C05408=1029.929,82.915,-98.730,168.536,44.482,158.314
C05409=1029.936,83.164,-98.749,168.538,44.480,158.314
C05410=1029.942,83.413,-98.767,168.540,44.479,158.314
C05411=1029.948,83.662,-98.785,168.542,44.477,158.313
C05412=1029.954,83.911,-98.804,168.545,44.474,158.313
C05413=1029.960,84.161,-98.821,168.547,44.472,158.313
C05414=1029.967,84.410,-98.840,168.550,44.470,158.313
C05415=1029.972,84.659,-98.859,168.552,44.468,158.313
C05416=1029.979,84.909,-98.877,168.555,44.466,158.313
C05417=1029.984,85.157,-98.896,168.557,44.465,158.312
C05418=1029.991,85.406,-98.914,168.559,44.463,158.312
C05419=1029.997,85.656,-98.932,168.561,44.460,158.312
C05420=1030.003,85.905,-98.951,168.564,44.458,158.312
C05421=1030.010,86.154,-98.969,168.567,44.456,158.312
C05422=1030.016,86.404,-98.988,168.569,44.454,158.312
C05423=1030.022,86.654,-99.007,168.572,44.452,158.312
C05424=1030.027,86.902,-99.025,168.573,44.451,158.311
C05425=1030.034,87.151,-99.044,168.576,44.448,158.311
C05426=1030.040,87.400,-99.062,168.578,44.446,158.311
C05427=1030.046,87.650,-99.080,168.581,44.444,158.311
C05428=1030.053,87.899,-99.099,168.583,44.442,158.311
C05429=1030.059,88.148,-99.117,168.586,44.440,158.311
C05430=1030.066,88.397,-99.136,168.588,44.438,158.310
C05431=1030.071,88.647,-99.155,168.591,44.436,158.310
C05432=1030.077,88.897,-99.173,168.593,44.434,158.310
C05433=1030.084,89.146,-99.192,168.595,44.432,158.310
C05434=1030.090,89.395,-99.211,168.598,44.430,158.310
C05435=1030.096,89.643,-99.229,168.600,44.428,158.309
C05436=1030.103,89.892,-99.247,168.603,44.426,158.309
C05437=1030.108,90.142,-99.267,168.605,44.424,158.309
C05438=1030.114,90.392,-99.285,168.608,44.422,158.309
C05439=1030.120,90.641,-99.304,168.609,44.420,158.309
C05440=1030.126,90.890,-99.323,168.612,44.418,158.309
C05441=1030.132,91.140,-99.342,168.615,44.416,158.309
C05442=1030.139,91.389,-99.360,168.617,44.414,158.308
C05443=1030.145,91.638,-99.379,168.620,44.412,158.308
C05444=1030.152,91.923,-99.401,168.622,44.410,158.308
C05445=1030.158,92.208,-99.422,168.625,44.408,158.308
C05446=1030.165,92.493,-99.444,168.627,44.406,158.308
C05447=1030.173,92.778,-99.466,168.631,44.404,158.308
C05448=1030.178,93.027,-99.485,168.633,44.402,158.308
C05449=1030.185,93.277,-99.504,168.635,44.400,158.307
C05450=1030.191,93.526,-99.523,168.637,44.398,158.307
C05451=1030.197,93.775,-99.541,168.640,44.396,158.307
C05452=1030.203,94.025,-99.561,168.642,44.394,158.307
C05453=1030.209,94.274,-99.579,168.645,44.392,158.307
C05454=1030.216,94.523,-99.598,168.648,44.390,158.307
C05455=1030.221,94.772,-99.617,168.650,44.388,158.306
C05456=1030.228,95.021,-99.636,168.652,44.386,158.306
C05457=1030.233,95.271,-99.655,168.654,44.384,158.306
C05458=1030.240,95.520,-99.674,168.657,44.382,158.306
C05459=1030.245,95.769,-99.693,168.660,44.380,158.306
C05460=1030.252,96.019,-99.712,168.662,44.378,158.306
C05461=1030.258,96.268,-99.730,168.664,44.376,158.305
C05462=1030.264,96.517,-99.750,168.667,44.374,158.305
C05463=1030.271,96.766,-99.769,168.669,44.372,158.305
C05464=1030.276,97.015,-99.788,168.671,44.370,158.305
C05465=1030.283,97.264,-99.807,168.674,44.368,158.305
C05466=1030.289,97.514,-99.826,168.676,44.366,158.305
C05467=1030.295,97.763,-99.845,168.679,44.365,158.305
C05468=1030.301,98.012,-99.864,168.682,44.363,158.304
C05469=1030.307,98.261,-99.883,168.684,44.361,158.304
C05470=1030.314,98.510,-99.901,168.687,44.358,158.304
C05471=1030.319,98.759,-99.921,168.688,44.356,158.304
C05472=1030.326,99.008,-99.940,168.691,44.354,158.304
C05473=1030.332,99.258,-99.959,168.693,44.353,158.304
C05474=1030.338,99.507,-99.978,168.696,44.351,158.303
C05475=1030.344,99.756,-99.997,168.698,44.349,158.303
C05476=1030.350,100.005,-100.016,168.701,44.347,158.303
C05477=1030.356,100.254,-100.036,168.704,44.345,158.303
C05478=1030.362,100.504,-100.055,168.706,44.343,158.303
C05479=1030.368,100.754,-100.074,168.708,44.341,158.303
C05480=1030.375,101.002,-100.094,168.710,44.339,158.303
C05481=1030.381,101.252,-100.113,168.713,44.337,158.302
C05482=1030.386,101.501,-100.132,168.715,44.335,158.302
C05483=1030.393,101.750,-100.152,168.718,44.334,158.302
C05484=1030.399,101.999,-100.171,168.721,44.332,158.302
C05485=1030.404,102.249,-100.190,168.723,44.330,158.302
C05486=1030.410,102.497,-100.210,168.725,44.328,158.302
C05487=1030.417,102.746,-100.229,168.727,44.326,158.302
C05488=1030.422,102.996,-100.248,168.730,44.324,158.301
C05489=1030.428,103.245,-100.268,168.733,44.322,158.301
C05490=1030.435,103.494,-100.287,168.735,44.320,158.301
C05491=1030.441,103.743,-100.307,168.738,44.318,158.301
C05492=1030.447,103.992,-100.326,168.740,44.316,158.301
C05493=1030.453,104.242,-100.345,168.742,44.315,158.301
C05494=1030.460,104.491,-100.365,168.744,44.313,158.301
C05495=1030.465,104.740,-100.384,168.747,44.311,158.300
C05496=1030.471,104.989,-100.404,168.749,44.308,158.300
C05497=1030.477,105.238,-100.423,168.752,44.306,158.300
C05498=1030.483,105.487,-100.442,168.755,44.304,158.300
C05499=1030.489,105.736,-100.462,168.757,44.303,158.300
C05500=1030.495,105.986,-100.481,168.760,44.301,158.300
C05501=1030.502,106.235,-100.501,168.761,44.299,158.299
C05502=1030.508,106.484,-100.520,168.764,44.297,158.299
C05503=1030.514,106.733,-100.540,168.767,44.295,158.299
C05504=1030.520,106.983,-100.559,168.769,44.293,158.299
C05505=1030.526,107.231,-100.579,168.772,44.291,158.299
C05506=1030.532,107.481,-100.598,168.774,44.289,158.299
C05507=1030.538,107.729,-100.618,168.777,44.287,158.299
C05508=1030.546,108.015,-100.640,168.779,44.285,158.298
C05509=1030.552,108.300,-100.662,168.782,44.283,158.298
C05510=1030.560,108.586,-100.685,168.785,44.281,158.298
C05511=1030.566,108.871,-100.707,168.788,44.278,158.298
C05512=1030.573,109.120,-100.726,168.790,44.276,158.298
C05513=1030.579,109.368,-100.746,168.793,44.274,158.298
C05514=1030.585,109.619,-100.766,168.796,44.272,158.297
C05515=1030.591,109.867,-100.786,168.798,44.271,158.297
C05516=1030.597,110.116,-100.805,168.801,44.269,158.297
C05517=1030.603,110.365,-100.825,168.803,44.267,158.297
C05518=1030.610,110.615,-100.844,168.805,44.265,158.297
C05519=1030.616,110.864,-100.864,168.807,44.263,158.297
C05520=1030.622,111.113,-100.884,168.810,44.261,158.297
C05521=1030.627,111.362,-100.903,168.813,44.259,158.296
C05522=1030.633,111.611,-100.923,168.815,44.257,158.296
C05523=1030.640,111.861,-100.944,168.818,44.255,158.296
C05524=1030.646,112.110,-100.963,168.820,44.253,158.296
C05525=1030.652,112.359,-100.983,168.823,44.252,158.296
C05526=1030.658,112.608,-101.003,168.826,44.250,158.296
C05527=1030.663,112.857,-101.022,168.828,44.248,158.296
C05528=1030.670,113.107,-101.042,168.830,44.246,158.295
C05529=1030.676,113.356,-101.062,168.832,44.244,158.295
C05530=1030.682,113.604,-101.082,168.835,44.242,158.295
C05531=1030.688,113.854,-101.102,168.838,44.241,158.295
C05532=1030.694,114.103,-101.122,168.840,44.239,158.295
C05533=1030.699,114.352,-101.142,168.843,44.237,158.295
C05534=1030.705,114.601,-101.162,168.845,44.235,158.295
C05535=1030.711,114.850,-101.182,168.847,44.234,158.294
C05536=1030.717,115.099,-101.202,168.850,44.232,158.294
C05537=1030.724,115.349,-101.222,168.852,44.230,158.294
C05538=1030.729,115.598,-101.242,168.855,44.228,158.294
C05539=1030.735,115.847,-101.262,168.858,44.227,158.294
C05540=1030.741,116.096,-101.282,168.860,44.225,158.294
C05541=1030.748,116.345,-101.303,168.863,44.223,158.294
C05542=1030.754,116.594,-101.323,168.865,44.221,158.294
C05543=1030.759,116.843,-101.343,168.867,44.219,158.293
C05544=1030.765,117.092,-101.363,168.870,44.217,158.293
C05545=1030.771,117.342,-101.383,168.872,44.215,158.293
C05546=1030.777,117.590,-101.403,168.875,44.213,158.293
C05547=1030.783,117.840,-101.423,168.878,44.212,158.293
C05548=1030.788,118.089,-101.443,168.880,44.210,158.293
C05549=1030.795,118.338,-101.464,168.883,44.208,158.293
C05550=1030.801,118.587,-101.484,168.885,44.206,158.293
C05551=1030.807,118.836,-101.503,168.888,44.204,158.293
C05552=1030.813,119.086,-101.524,168.889,44.203,158.292
C05553=1030.819,119.335,-101.544,168.892,44.201,158.292
C05554=1030.825,119.584,-101.564,168.895,44.199,158.292
C05555=1030.831,119.833,-101.585,168.897,44.197,158.292
C05556=1030.837,120.082,-101.605,168.900,44.195,158.292
C05557=1030.843,120.331,-101.625,168.903,44.194,158.292
C05558=1030.849,120.581,-101.645,168.905,44.192,158.292
C05559=1030.855,120.829,-101.665,168.908,44.190,158.291
C05560=1030.861,121.078,-101.685,168.910,44.188,158.291
C05561=1030.867,121.328,-101.706,168.913,44.186,158.291
C05562=1030.873,121.577,-101.726,168.916,44.184,158.291
C05563=1030.879,121.826,-101.746,168.918,44.182,158.291
C05564=1030.886,122.075,-101.767,168.920,44.181,158.291
C05565=1030.892,122.324,-101.787,168.922,44.179,158.291
C05566=1030.897,122.573,-101.807,168.925,44.177,158.290
C05567=1030.904,122.822,-101.828,168.927,44.175,158.290
C05568=1030.910,123.071,-101.848,168.930,44.173,158.290
C05569=1030.916,123.320,-101.868,168.933,44.172,158.290
C05570=1030.922,123.569,-101.889,168.935,44.170,158.290
C05571=1030.928,123.818,-101.909,168.938,44.168,158.290
C05572=1030.935,124.104,-101.933,168.940,44.165,158.290
C05573=1030.942,124.388,-101.955,168.944,44.163,158.290
C05574=1030.949,124.673,-101.979,168.947,44.161,158.289
C05575=1030.956,124.959,-102.003,168.950,44.159,158.289
C05576=1030.962,125.208,-102.023,168.953,44.157,158.289
C05577=1030.968,125.457,-102.043,168.955,44.156,158.289
C05578=1030.974,125.706,-102.063,168.958,44.154,158.289
C05579=1030.980,125.955,-102.083,168.960,44.152,158.289
C05580=1030.986,126.205,-102.104,168.962,44.150,158.289
C05581=1030.993,126.453,-102.124,168.965,44.148,158.288
C05582=1030.999,126.702,-102.145,168.967,44.146,158.288
C05583=1031.004,126.951,-102.165,168.970,44.144,158.288
C05584=1031.011,127.201,-102.186,168.973,44.142,158.288
C05585=1031.017,127.450,-102.206,168.975,44.141,158.288
C05586=1031.024,127.699,-102.227,168.978,44.139,158.288
C05587=1031.029,127.948,-102.247,168.980,44.137,158.288
C05588=1031.036,128.197,-102.267,168.983,44.135,158.287
C05589=1031.042,128.446,-102.287,168.985,44.133,158.287
C05590=1031.049,128.695,-102.308,168.988,44.131,158.287
C05591=1031.054,128.944,-102.329,168.991,44.129,158.287
C05592=1031.060,129.194,-102.349,168.993,44.128,158.287
C05593=1031.066,129.442,-102.369,168.996,44.126,158.287
C05594=1031.073,129.692,-102.391,168.999,44.124,158.287
C05595=1031.079,129.940,-102.411,169.001,44.122,158.287
C05596=1031.085,130.190,-102.431,169.004,44.120,158.286
C05597=1031.092,130.438,-102.452,169.006,44.118,158.286
C05598=1031.097,130.688,-102.473,169.009,44.116,158.286
C05599=1031.103,130.937,-102.493,169.012,44.115,158.286
C05600=1031.110,131.186,-102.514,169.014,44.113,158.286
C05601=1031.115,131.435,-102.535,169.017,44.111,158.286
C05602=1031.122,131.684,-102.556,169.020,44.110,158.286
C05603=1031.127,131.933,-102.577,169.022,44.108,158.286
C05604=1031.134,132.183,-102.597,169.025,44.106,158.285
C05605=1031.139,132.431,-102.618,169.027,44.104,158.285
C05606=1031.146,132.681,-102.638,169.030,44.102,158.285
C05607=1031.151,132.929,-102.660,169.033,44.101,158.285
C05608=1031.157,133.179,-102.681,169.035,44.099,158.285
C05609=1031.163,133.427,-102.701,169.038,44.097,158.285
C05610=1031.169,133.677,-102.722,169.041,44.095,158.285
C05611=1031.176,133.925,-102.743,169.043,44.093,158.285
C05612=1031.181,134.175,-102.764,169.046,44.091,158.284
C05613=1031.187,134.423,-102.785,169.049,44.090,158.284
C05614=1031.194,134.673,-102.805,169.051,44.088,158.284
C05615=1031.199,134.922,-102.827,169.054,44.086,158.284
C05616=1031.206,135.170,-102.848,169.056,44.084,158.284
C05617=1031.211,135.420,-102.868,169.059,44.082,158.284
C05618=1031.217,135.669,-102.890,169.062,44.081,158.284
C05619=1031.224,135.918,-102.910,169.064,44.079,158.284
C05620=1031.230,136.167,-102.932,169.067,44.077,158.284
C05621=1031.236,136.416,-102.952,169.069,44.075,158.283
C05622=1031.242,136.665,-102.973,169.072,44.074,158.283
C05623=1031.248,136.914,-102.995,169.075,44.072,158.283
C05624=1031.255,137.163,-103.015,169.077,44.070,158.283
C05625=1031.260,137.412,-103.036,169.080,44.069,158.283
C05626=1031.266,137.661,-103.058,169.083,44.067,158.283
C05627=1031.272,137.910,-103.078,169.085,44.065,158.283
C05628=1031.278,138.159,-103.100,169.088,44.064,158.283
C05629=1031.284,138.408,-103.121,169.091,44.062,158.283
C05630=1031.290,138.658,-103.142,169.093,44.060,158.282
C05631=1031.297,138.906,-103.163,169.096,44.058,158.282
C05632=1031.302,139.155,-103.184,169.099,44.057,158.282
C05633=1031.308,139.405,-103.205,169.101,44.055,158.282
C05634=1031.314,139.654,-103.227,169.104,44.053,158.282
C05635=1031.320,139.902,-103.248,169.106,44.051,158.282
C05636=1031.327,140.187,-103.272,169.110,44.049,158.282
C05637=1031.334,140.473,-103.296,169.113,44.048,158.282
C05638=1031.341,140.758,-103.321,169.115,44.046,158.282
C05639=1031.347,141.042,-103.345,169.119,44.044,158.282
C05640=1031.354,141.291,-103.367,169.122,44.042,158.281
C05641=1031.360,141.541,-103.387,169.124,44.040,158.281
C05642=1031.365,141.789,-103.409,169.127,44.039,158.281
C05643=1031.371,142.039,-103.430,169.130,44.037,158.281
C05644=1031.378,142.287,-103.451,169.132,44.035,158.281
C05645=1031.384,142.536,-103.473,169.135,44.033,158.281
C05646=1031.390,142.785,-103.494,169.138,44.032,158.281
C05647=1031.396,143.034,-103.516,169.140,44.030,158.281
C05648=1031.401,143.283,-103.537,169.143,44.028,158.281
C05649=1031.407,143.533,-103.558,169.146,44.027,158.281
C05650=1031.414,143.782,-103.580,169.148,44.025,158.280
C05651=1031.420,144.030,-103.600,169.151,44.023,158.280
C05652=1031.426,144.279,-103.622,169.153,44.021,158.280
C05653=1031.432,144.528,-103.644,169.156,44.020,158.280
C05654=1031.438,144.778,-103.665,169.159,44.018,158.280
C05655=1031.444,145.026,-103.687,169.161,44.016,158.280
C05656=1031.450,145.275,-103.708,169.165,44.015,158.280
C05657=1031.456,145.525,-103.730,169.168,44.013,158.280
C05658=1031.462,145.773,-103.751,169.170,44.011,158.280
C05659=1031.469,146.022,-103.772,169.173,44.009,158.279
C05660=1031.475,146.271,-103.794,169.176,44.008,158.279
C05661=1031.481,146.520,-103.815,169.178,44.006,158.279
C05662=1031.487,146.769,-103.837,169.181,44.004,158.279
C05663=1031.493,147.018,-103.858,169.184,44.003,158.279
C05664=1031.499,147.267,-103.880,169.186,44.001,158.279
C05665=1031.505,147.517,-103.902,169.189,43.999,158.279
C05666=1031.511,147.765,-103.923,169.192,43.998,158.279
C05667=1031.517,148.014,-103.945,169.194,43.996,158.279
C05668=1031.522,148.264,-103.967,169.197,43.994,158.279
C05669=1031.528,148.513,-103.988,169.200,43.993,158.279
C05670=1031.534,148.761,-104.010,169.202,43.991,158.278
C05671=1031.540,149.011,-104.031,169.205,43.990,158.278
C05672=1031.546,149.260,-104.053,169.209,43.987,158.278
C05673=1031.553,149.508,-104.075,169.212,43.986,158.278
C05674=1031.558,149.757,-104.097,169.214,43.984,158.278
C05675=1031.565,150.006,-104.118,169.217,43.982,158.278
C05676=1031.571,150.255,-104.140,169.220,43.981,158.278
C05677=1031.576,150.505,-104.162,169.222,43.979,158.278
C05678=1031.582,150.753,-104.184,169.225,43.977,158.278
C05679=1031.588,151.002,-104.206,169.228,43.976,158.278
C05680=1031.594,151.251,-104.227,169.230,43.974,158.278
C05681=1031.600,151.500,-104.249,169.233,43.973,158.278
C05682=1031.607,151.750,-104.271,169.236,43.971,158.277
C05683=1031.613,151.998,-104.293,169.238,43.969,158.277
C05684=1031.618,152.247,-104.315,169.242,43.968,158.277
C05685=1031.624,152.496,-104.336,169.245,43.966,158.277
C05686=1031.630,152.745,-104.358,169.248,43.965,158.277
C05687=1031.637,152.994,-104.380,169.250,43.963,158.277
C05688=1031.643,153.243,-104.402,169.253,43.962,158.277
C05689=1031.649,153.492,-104.424,169.256,43.960,158.277
C05690=1031.655,153.740,-104.446,169.258,43.958,158.277
C05691=1031.660,153.990,-104.468,169.261,43.957,158.277
C05692=1031.666,154.239,-104.490,169.264,43.955,158.277
C05693=1031.673,154.488,-104.512,169.266,43.954,158.277
C05694=1031.678,154.737,-104.534,169.270,43.952,158.276
C05695=1031.685,154.986,-104.556,169.273,43.950,158.276
C05696=1031.690,155.234,-104.578,169.275,43.948,158.276
C05697=1031.697,155.483,-104.599,169.278,43.947,158.276
C05698=1031.702,155.732,-104.622,169.281,43.945,158.276
C05699=1031.708,155.982,-104.644,169.284,43.944,158.276
C05700=1031.715,156.266,-104.670,169.287,43.942,158.276
C05701=1031.722,156.551,-104.695,169.290,43.940,158.276
C05702=1031.730,156.835,-104.720,169.293,43.938,158.276
C05703=1031.736,157.120,-104.745,169.296,43.937,158.276
C05704=1031.742,157.369,-104.768,169.300,43.935,158.276
C05705=1031.748,157.618,-104.789,169.303,43.934,158.276
C05706=1031.754,157.867,-104.812,169.305,43.932,158.276
C05707=1031.761,158.116,-104.833,169.308,43.930,158.276
C05708=1031.766,158.364,-104.856,169.311,43.929,158.275
C05709=1031.772,158.614,-104.877,169.314,43.927,158.275
C05710=1031.778,158.862,-104.900,169.316,43.925,158.275
C05711=1031.784,159.112,-104.922,169.320,43.923,158.275
C05712=1031.790,159.360,-104.944,169.323,43.922,158.275
C05713=1031.796,159.609,-104.966,169.325,43.920,158.275
C05714=1031.802,159.858,-104.989,169.328,43.919,158.275
C05715=1031.808,160.107,-105.012,169.331,43.918,158.275
C05716=1031.814,160.356,-105.034,169.333,43.916,158.275
C05717=1031.820,160.605,-105.057,169.336,43.915,158.275
C05718=1031.826,160.854,-105.079,169.339,43.913,158.275
C05719=1031.831,161.104,-105.102,169.342,43.912,158.275
C05720=1031.837,161.352,-105.124,169.345,43.910,158.275
C05721=1031.843,161.601,-105.147,169.348,43.909,158.275
C05722=1031.848,161.849,-105.170,169.351,43.908,158.275
C05723=1031.854,162.099,-105.192,169.354,43.906,158.275
C05724=1031.860,162.348,-105.214,169.357,43.905,158.275
C05725=1031.866,162.596,-105.237,169.359,43.903,158.275
C05726=1031.872,162.845,-105.260,169.362,43.902,158.275
C05727=1031.877,163.094,-105.283,169.365,43.900,158.274
C05728=1031.884,163.343,-105.305,169.368,43.899,158.274
C05729=1031.889,163.592,-105.328,169.371,43.898,158.275
C05730=1031.895,163.841,-105.351,169.374,43.896,158.274
C05731=1031.901,164.090,-105.373,169.377,43.895,158.274
C05732=1031.907,164.339,-105.396,169.380,43.893,158.274
C05733=1031.913,164.588,-105.419,169.382,43.892,158.274
C05734=1031.918,164.837,-105.441,169.385,43.890,158.274
C05735=1031.924,165.086,-105.464,169.388,43.889,158.274
C05736=1031.931,165.335,-105.486,169.392,43.888,158.274
C05737=1031.936,165.583,-105.509,169.395,43.886,158.274
C05738=1031.942,165.832,-105.532,169.397,43.884,158.274
C05739=1031.948,166.081,-105.555,169.400,43.883,158.274
C05740=1031.954,166.330,-105.577,169.403,43.882,158.274
C05741=1031.960,166.579,-105.600,169.405,43.880,158.274
C05742=1031.966,166.828,-105.623,169.409,43.879,158.274
C05743=1031.971,167.077,-105.646,169.412,43.878,158.274
C05744=1031.978,167.325,-105.669,169.415,43.876,158.274
C05745=1031.983,167.575,-105.691,169.417,43.874,158.274
C05746=1031.989,167.824,-105.714,169.420,43.873,158.274
C05747=1031.995,168.072,-105.737,169.424,43.872,158.274
C05748=1032.001,168.321,-105.759,169.427,43.870,158.274
C05749=1032.007,168.570,-105.782,169.429,43.869,158.274
C05750=1032.013,168.819,-105.805,169.432,43.867,158.274
C05751=1032.018,169.068,-105.828,169.435,43.866,158.274
C05752=1032.025,169.317,-105.851,169.439,43.864,158.274
C05753=1032.031,169.566,-105.874,169.442,43.863,158.274
C05754=1032.037,169.814,-105.897,169.444,43.862,158.274
C05755=1032.043,170.063,-105.920,169.447,43.861,158.274
C05756=1032.049,170.312,-105.943,169.450,43.859,158.273
C05757=1032.055,170.561,-105.966,169.454,43.857,158.273
C05758=1032.061,170.809,-105.988,169.456,43.856,158.273
C05759=1032.067,171.058,-106.011,169.459,43.855,158.273
C05760=1032.073,171.308,-106.035,169.462,43.853,158.273
C05761=1032.079,171.557,-106.058,169.466,43.852,158.273
C05762=1032.085,171.805,-106.080,169.468,43.850,158.273
C05763=1032.091,172.054,-106.103,169.471,43.849,158.273
C05764=1032.098,172.338,-106.129,169.475,43.847,158.273
C05765=1032.104,172.623,-106.156,169.479,43.846,158.273
C05766=1032.111,172.907,-106.182,169.481,43.844,158.273
C05767=1032.119,173.191,-106.208,169.485,43.842,158.273
C05768=1032.124,173.439,-106.231,169.488,43.841,158.273
C05769=1032.130,173.688,-106.254,169.492,43.839,158.273
C05770=1032.136,173.938,-106.278,169.494,43.838,158.273
C05771=1032.143,174.187,-106.300,169.497,43.837,158.273
C05772=1032.149,174.435,-106.324,169.500,43.835,158.273
C05773=1032.155,174.684,-106.347,169.504,43.833,158.273
C05774=1032.160,174.933,-106.370,169.506,43.832,158.273
C05775=1032.167,175.182,-106.393,169.509,43.831,158.273
C05776=1032.173,175.431,-106.415,169.513,43.830,158.273
C05777=1032.179,175.679,-106.439,169.516,43.828,158.273
C05778=1032.185,175.928,-106.462,169.519,43.826,158.273
C05779=1032.191,176.178,-106.485,169.522,43.825,158.273
C05780=1032.197,176.426,-106.509,169.525,43.824,158.273
C05781=1032.203,176.675,-106.532,169.528,43.822,158.273
C05782=1032.210,176.924,-106.554,169.531,43.821,158.273
C05783=1032.216,177.173,-106.577,169.534,43.819,158.273
C05784=1032.222,177.421,-106.601,169.537,43.818,158.273
C05785=1032.228,177.670,-106.624,169.540,43.817,158.273
C05786=1032.234,177.920,-106.647,169.544,43.815,158.273
C05787=1032.241,178.168,-106.670,169.547,43.814,158.273
C05788=1032.247,178.417,-106.693,169.549,43.812,158.273
C05789=1032.253,178.666,-106.717,169.553,43.811,158.273
C05790=1032.259,178.914,-106.740,169.556,43.810,158.273
C05791=1032.265,179.163,-106.763,169.559,43.808,158.272
C05792=1032.271,179.412,-106.787,169.562,43.806,158.273
C05793=1032.278,179.661,-106.810,169.565,43.805,158.273
C05794=1032.284,179.909,-106.833,169.569,43.804,158.273
C05795=1032.290,180.159,-106.857,169.572,43.803,158.273
C05796=1032.296,180.408,-106.880,169.574,43.801,158.272
C05797=1032.302,180.656,-106.903,169.578,43.799,158.272
C05798=1032.308,180.906,-106.927,169.581,43.798,158.272
C05799=1032.315,181.154,-106.950,169.584,43.797,158.272
C05800=1032.321,181.403,-106.973,169.588,43.796,158.272
C05801=1032.327,181.651,-106.997,169.590,43.794,158.272
C05802=1032.333,181.900,-107.020,169.594,43.792,158.272
C05803=1032.340,182.149,-107.044,169.597,43.791,158.272
C05804=1032.345,182.398,-107.066,169.600,43.790,158.272
C05805=1032.352,182.647,-107.091,169.604,43.788,158.272
C05806=1032.359,182.896,-107.113,169.606,43.787,158.272
C05807=1032.364,183.145,-107.137,169.610,43.785,158.272
C05808=1032.370,183.393,-107.161,169.613,43.784,158.272
C05809=1032.376,183.642,-107.184,169.616,43.783,158.272
C05810=1032.381,183.891,-107.208,169.620,43.782,158.272
C05811=1032.388,184.140,-107.232,169.623,43.781,158.272
C05812=1032.393,184.388,-107.257,169.625,43.780,158.272
C05813=1032.400,184.638,-107.280,169.628,43.778,158.272
C05814=1032.406,184.886,-107.304,169.632,43.777,158.272
C05815=1032.411,185.135,-107.328,169.635,43.776,158.272
C05816=1032.418,185.384,-107.352,169.638,43.775,158.273
C05817=1032.423,185.632,-107.376,169.642,43.774,158.273
C05818=1032.429,185.881,-107.400,169.645,43.773,158.273
C05819=1032.435,186.131,-107.424,169.647,43.771,158.273
C05820=1032.441,186.379,-107.447,169.651,43.770,158.273
C05821=1032.447,186.628,-107.472,169.654,43.769,158.273
C05822=1032.453,186.876,-107.496,169.658,43.768,158.273
C05823=1032.459,187.125,-107.519,169.661,43.767,158.273
C05824=1032.465,187.374,-107.544,169.664,43.766,158.273
C05825=1032.471,187.622,-107.568,169.668,43.764,158.273
C05826=1032.477,187.872,-107.592,169.670,43.763,158.273
C05827=1032.482,188.120,-107.615,169.673,43.762,158.273
C05828=1032.489,188.404,-107.643,169.677,43.760,158.273
C05829=1032.496,188.687,-107.671,169.681,43.759,158.273
C05830=1032.502,188.972,-107.698,169.685,43.758,158.273
C05831=1032.510,189.256,-107.726,169.689,43.757,158.273
C05832=1032.516,189.504,-107.749,169.692,43.756,158.273
C05833=1032.521,189.753,-107.774,169.695,43.754,158.273
C05834=1032.528,190.002,-107.798,169.698,43.753,158.273
C05835=1032.533,190.250,-107.822,169.701,43.752,158.273
C05836=1032.539,190.499,-107.846,169.705,43.751,158.273
C05837=1032.545,190.748,-107.870,169.708,43.750,158.273
C05838=1032.551,190.997,-107.894,169.712,43.748,158.273
C05839=1032.557,191.246,-107.919,169.715,43.747,158.273
C05840=1032.563,191.494,-107.942,169.718,43.746,158.273
C05841=1032.570,191.743,-107.966,169.721,43.745,158.274
C05842=1032.576,191.991,-107.991,169.724,43.744,158.274
C05843=1032.582,192.240,-108.015,169.728,43.743,158.274
C05844=1032.588,192.489,-108.040,169.731,43.741,158.274
C05845=1032.594,192.738,-108.064,169.735,43.740,158.274
C05846=1032.599,192.986,-108.088,169.738,43.739,158.274
C05847=1032.606,193.235,-108.112,169.742,43.738,158.274
C05848=1032.612,193.485,-108.137,169.744,43.737,158.274
C05849=1032.618,193.733,-108.160,169.748,43.735,158.274
C05850=1032.624,193.982,-108.186,169.751,43.735,158.274
C05851=1032.630,194.230,-108.209,169.755,43.733,158.274
C05852=1032.636,194.479,-108.234,169.758,43.732,158.274
C05853=1032.643,194.728,-108.258,169.761,43.731,158.274
C05854=1032.648,194.977,-108.282,169.765,43.730,158.274
C05855=1032.655,195.225,-108.307,169.768,43.729,158.274
C05856=1032.660,195.474,-108.331,169.772,43.728,158.274
C05857=1032.667,195.723,-108.355,169.774,43.726,158.274
C05858=1032.673,195.972,-108.380,169.778,43.726,158.274
C05859=1032.679,196.220,-108.404,169.781,43.724,158.274
C05860=1032.685,196.469,-108.429,169.785,43.723,158.274
C05861=1032.692,196.718,-108.453,169.788,43.722,158.274
C05862=1032.697,196.967,-108.477,169.792,43.721,158.275
C05863=1032.704,197.215,-108.502,169.795,43.720,158.275
C05864=1032.710,197.464,-108.527,169.799,43.718,158.275
C05865=1032.716,197.712,-108.550,169.803,43.718,158.275
C05866=1032.722,197.961,-108.576,169.805,43.716,158.275
C05867=1032.729,198.210,-108.600,169.809,43.715,158.275
C05868=1032.735,198.459,-108.624,169.812,43.715,158.275
C05869=1032.741,198.707,-108.649,169.816,43.713,158.275
C05870=1032.747,198.956,-108.673,169.819,43.712,158.275
C05871=1032.754,199.205,-108.698,169.823,43.711,158.275
C05872=1032.760,199.454,-108.723,169.826,43.710,158.275
C05873=1032.766,199.702,-108.746,169.830,43.709,158.275
C05874=1032.772,199.951,-108.772,169.832,43.707,158.275
C05875=1032.779,200.200,-108.796,169.837,43.707,158.275
C05876=1032.785,200.449,-108.821,169.840,43.705,158.275
C05877=1032.790,200.697,-108.845,169.843,43.705,158.276
C05878=1032.796,200.946,-108.870,169.847,43.703,158.276
C05879=1032.803,201.195,-108.895,169.850,43.703,158.276
C05880=1032.809,201.443,-108.920,169.854,43.701,158.276
C05881=1032.815,201.691,-108.945,169.857,43.701,158.276
C05882=1032.821,201.941,-108.969,169.861,43.699,158.276
C05883=1032.827,202.189,-108.995,169.864,43.699,158.276
C05884=1032.833,202.439,-109.019,169.868,43.697,158.276
C05885=1032.838,202.687,-109.044,169.871,43.697,158.276
C05886=1032.845,202.935,-109.070,169.875,43.695,158.276
C05887=1032.851,203.184,-109.094,169.879,43.695,158.276
C05888=1032.858,203.433,-109.119,169.882,43.693,158.276
C05889=1032.864,203.682,-109.144,169.886,43.693,158.277
C05890=1032.869,203.930,-109.169,169.888,43.692,158.277
C05891=1032.875,204.179,-109.194,169.893,43.691,158.277
C05892=1032.901,205.228,-109.300,170.230,43.795,158.327
C05893=1032.911,205.577,-109.337,170.234,43.794,158.327
C05894=1032.921,205.926,-109.374,170.237,43.795,158.327
C05895=1032.930,206.275,-109.410,170.241,43.794,158.328
C05896=1032.940,206.624,-109.448,170.244,43.794,158.328
C05897=1032.946,206.873,-109.475,170.246,43.794,158.328
C05898=1032.953,207.121,-109.501,170.249,43.793,158.328
C05899=1032.960,207.370,-109.527,170.251,43.793,158.328
C05900=1032.966,207.618,-109.553,170.255,43.793,158.329
C05901=1032.973,207.867,-109.580,170.257,43.793,158.329
C05902=1032.980,208.116,-109.606,170.260,43.793,158.329
C05903=1032.986,208.364,-109.633,170.262,43.792,158.329
C05904=1032.994,208.612,-109.659,170.264,43.793,158.329
C05905=1032.999,208.861,-109.686,170.267,43.792,158.330
C05906=1033.006,209.110,-109.712,170.270,43.792,158.330
C05907=1033.014,209.358,-109.738,170.273,43.792,158.330
C05908=1033.020,209.606,-109.765,170.275,43.792,158.330
C05909=1033.027,209.855,-109.792,170.278,43.791,158.330
C05910=1033.034,210.104,-109.819,170.280,43.792,158.331
C05911=1033.040,210.352,-109.845,170.282,43.791,158.331
C05912=1033.047,210.601,-109.872,170.285,43.791,158.331
C05913=1033.054,210.849,-109.898,170.287,43.791,158.331
C05914=1033.061,211.097,-109.925,170.291,43.790,158.331
C05915=1033.067,211.346,-109.952,170.293,43.791,158.331
C05916=1033.074,211.595,-109.978,170.296,43.791,158.332
C05917=1033.080,211.843,-110.005,170.298,43.790,158.332
C05918=1033.087,212.091,-110.032,170.301,43.790,158.332
C05919=1033.093,212.340,-110.059,170.303,43.790,158.332
C05920=1033.100,212.588,-110.085,170.307,43.790,158.332
C05921=1033.107,212.837,-110.113,170.309,43.790,158.333
C05922=1033.113,213.085,-110.139,170.311,43.790,158.333
C05923=1033.120,213.334,-110.166,170.314,43.789,158.333
C05924=1033.127,213.582,-110.193,170.316,43.790,158.333
C05925=1033.134,213.831,-110.220,170.319,43.790,158.333
C05926=1033.140,214.079,-110.246,170.321,43.789,158.334
C05927=1033.147,214.328,-110.274,170.325,43.789,158.334
C05928=1033.154,214.576,-110.300,170.327,43.789,158.334
C05929=1033.160,214.825,-110.327,170.330,43.789,158.334
C05930=1033.167,215.073,-110.354,170.332,43.789,158.334
C05931=1033.173,215.322,-110.381,170.335,43.789,158.335
C05932=1033.181,215.570,-110.408,170.338,43.789,158.335
C05933=1033.187,215.818,-110.435,170.341,43.788,158.335
C05934=1033.194,216.067,-110.461,170.343,43.789,158.335
C05935=1033.200,216.316,-110.489,170.346,43.788,158.335
C05936=1033.208,216.564,-110.516,170.348,43.788,158.336
C05937=1033.214,216.812,-110.543,170.351,43.788,158.336
C05938=1033.221,217.061,-110.569,170.353,43.788,158.336
C05939=1033.227,217.309,-110.597,170.357,43.788,158.336
C05940=1033.235,217.558,-110.623,170.359,43.788,158.336
C05941=1033.241,217.806,-110.651,170.362,43.788,158.337
C05942=1033.248,218.054,-110.677,170.364,43.787,158.337
C05943=1033.254,218.303,-110.705,170.367,43.787,158.337
C05944=1033.262,218.552,-110.731,170.369,43.787,158.337
C05945=1033.268,218.800,-110.759,170.373,43.787,158.337
C05946=1033.275,219.048,-110.785,170.375,43.787,158.338
C05947=1033.281,219.297,-110.813,170.378,43.787,158.338
C05948=1033.289,219.545,-110.839,170.380,43.787,158.338
C05949=1033.297,219.900,-110.878,170.384,43.787,158.338
C05950=1033.307,220.255,-110.917,170.389,43.787,158.339
C05951=1033.317,220.609,-110.957,170.392,43.787,158.339
C05952=1033.326,220.964,-110.996,170.396,43.787,158.339
C05953=1033.333,221.213,-111.023,170.398,43.786,158.339
C05954=1033.339,221.461,-111.050,170.401,43.786,158.340
C05955=1033.346,221.710,-111.078,170.404,43.787,158.340
C05956=1033.353,221.958,-111.105,170.407,43.786,158.340
C05957=1033.359,222.207,-111.132,170.410,43.786,158.340
C05958=1033.366,222.455,-111.160,170.412,43.786,158.341
C05959=1033.372,222.703,-111.187,170.416,43.786,158.341
C05960=1033.379,222.951,-111.215,170.418,43.786,158.341
C05961=1033.386,223.200,-111.241,170.421,43.786,158.341
C05962=1033.393,223.449,-111.269,170.423,43.786,158.342
C05963=1033.399,223.697,-111.297,170.426,43.786,158.342
C05964=1033.406,223.945,-111.324,170.428,43.786,158.342
C05965=1033.413,224.194,-111.352,170.432,43.786,158.342
C05966=1033.420,224.443,-111.378,170.435,43.786,158.343
C05967=1033.426,224.690,-111.406,170.437,43.786,158.343
C05968=1033.432,224.939,-111.433,170.440,43.786,158.343
C05969=1033.439,225.187,-111.461,170.442,43.786,158.343
C05970=1033.446,225.436,-111.489,170.445,43.785,158.343
C05971=1033.453,225.684,-111.515,170.448,43.786,158.344
C05972=1033.460,225.933,-111.543,170.451,43.786,158.344
C05973=1033.466,226.181,-111.571,170.454,43.786,158.344
C05974=1033.473,226.430,-111.599,170.456,43.785,158.344
C05975=1033.480,226.678,-111.626,170.460,43.786,158.344
C05976=1033.486,226.927,-111.654,170.462,43.786,158.345
C05977=1033.494,227.175,-111.681,170.465,43.785,158.345
C05978=1033.500,227.423,-111.709,170.468,43.785,158.345
C05979=1033.507,227.672,-111.737,170.470,43.785,158.345
C05980=1033.514,227.920,-111.764,170.474,43.786,158.346
C05981=1033.520,228.168,-111.792,170.476,43.785,158.346
C05982=1033.527,228.416,-111.819,170.479,43.785,158.346
C05983=1033.533,228.665,-111.847,170.482,43.785,158.346
C05984=1033.540,228.913,-111.875,170.484,43.786,158.347
C05985=1033.547,229.162,-111.903,170.488,43.786,158.347
C05986=1033.553,229.410,-111.930,170.490,43.786,158.347
C05987=1033.560,229.659,-111.958,170.493,43.785,158.347
C05988=1033.567,229.907,-111.986,170.496,43.785,158.348
C05989=1033.573,230.155,-112.014,170.498,43.786,158.348
C05990=1033.580,230.404,-112.041,170.502,43.786,158.348
C05991=1033.587,230.652,-112.069,170.504,43.786,158.348
C05992=1033.593,230.901,-112.097,170.507,43.786,158.349
C05993=1033.600,231.149,-112.125,170.510,43.785,158.349
C05994=1033.607,231.397,-112.153,170.513,43.786,158.349
C05995=1033.613,231.646,-112.181,170.516,43.786,158.349
C05996=1033.620,231.894,-112.209,170.519,43.786,158.350
C05997=1033.626,232.143,-112.237,170.521,43.786,158.350
C05998=1033.633,232.390,-112.265,170.525,43.786,158.350
C05999=1033.640,232.639,-112.293,170.527,43.786,158.350
C06000=1033.646,232.888,-112.321,170.530,43.786,158.351
C06001=1033.653,233.136,-112.349,170.533,43.786,158.351
C06002=1033.659,233.385,-112.377,170.536,43.787,158.351
C06003=1033.666,233.632,-112.405,170.539,43.787,158.351
C06004=1033.673,233.881,-112.433,170.542,43.786,158.352
C06005=1033.682,234.228,-112.473,170.545,43.787,158.352
C06006=1033.691,234.575,-112.512,170.550,43.787,158.352
C06007=1033.700,234.923,-112.551,170.554,43.786,158.353
C06008=1033.709,235.270,-112.590,170.557,43.787,158.353
C06009=1033.716,235.518,-112.618,170.561,43.787,158.353
C06010=1033.724,235.767,-112.646,170.564,43.787,158.354
C06011=1033.730,236.015,-112.674,170.566,43.787,158.354
C06012=1033.737,236.263,-112.703,170.569,43.787,158.354
C06013=1033.743,236.512,-112.731,170.573,43.787,158.354
C06014=1033.750,236.760,-112.759,170.576,43.787,158.355
C06015=1033.757,237.008,-112.787,170.578,43.787,158.355
C06016=1033.763,237.257,-112.815,170.581,43.787,158.355
C06017=1033.770,237.505,-112.844,170.585,43.787,158.356
C06018=1033.777,237.753,-112.872,170.587,43.788,158.356
C06019=1033.784,238.002,-112.900,170.590,43.788,158.356
C06020=1033.790,238.250,-112.929,170.593,43.788,158.356
C06021=1033.797,238.498,-112.957,170.596,43.788,158.357
C06022=1033.804,238.747,-112.985,170.599,43.788,158.357
C06023=1033.810,238.995,-113.014,170.602,43.788,158.357
C06024=1033.817,239.243,-113.042,170.605,43.788,158.357
C06025=1033.824,239.491,-113.070,170.608,43.788,158.358
C06026=1033.831,239.740,-113.098,170.611,43.788,158.358
C06027=1033.837,239.988,-113.127,170.614,43.788,158.358
C06028=1033.844,240.237,-113.155,170.616,43.789,158.359
C06029=1033.851,240.484,-113.183,170.620,43.789,158.359
C06030=1033.857,240.733,-113.212,170.623,43.789,158.359
C06031=1033.864,240.981,-113.240,170.626,43.789,158.359
C06032=1033.870,241.229,-113.269,170.628,43.789,158.360
C06033=1033.878,241.478,-113.298,170.632,43.789,158.360
C06034=1033.884,241.726,-113.326,170.635,43.789,158.360
C06035=1033.891,241.974,-113.355,170.637,43.789,158.360
C06036=1033.897,242.222,-113.384,170.641,43.790,158.361
C06037=1033.904,242.470,-113.412,170.644,43.790,158.361
C06038=1033.910,242.720,-113.441,170.647,43.790,158.361
C06039=1033.917,242.968,-113.470,170.649,43.790,158.362
C06040=1033.924,243.216,-113.498,170.653,43.791,158.362
C06041=1033.930,243.464,-113.528,170.656,43.791,158.362
C06042=1033.937,243.712,-113.555,170.658,43.791,158.363
C06043=1033.943,243.961,-113.585,170.662,43.791,158.363
C06044=1033.950,244.209,-113.613,170.665,43.792,158.363
C06045=1033.957,244.457,-113.642,170.668,43.792,158.364
C06046=1033.964,244.705,-113.671,170.671,43.792,158.364
C06047=1033.970,244.954,-113.699,170.674,43.792,158.364
C06048=1033.976,245.202,-113.728,170.677,43.792,158.364
C06049=1033.983,245.451,-113.757,170.681,43.793,158.365
C06050=1033.989,245.699,-113.786,170.683,43.793,158.365
C06051=1033.996,245.946,-113.815,170.686,43.793,158.365
C06052=1034.002,246.195,-113.844,170.689,43.793,158.366
C06053=1034.009,246.443,-113.873,170.692,43.794,158.366
C06054=1034.015,246.692,-113.902,170.695,43.794,158.366
C06055=1034.022,246.940,-113.931,170.698,43.794,158.367
C06056=1034.029,247.188,-113.960,170.702,43.794,158.367
C06057=1034.035,247.436,-113.989,170.704,43.795,158.367
C06058=1034.042,247.684,-114.018,170.707,43.795,158.368
C06059=1034.048,247.933,-114.047,170.711,43.795,158.368
C06060=1034.054,248.181,-114.076,170.714,43.795,158.368
C06061=1034.063,248.522,-114.116,170.718,43.795,158.369
C06062=1034.073,248.863,-114.156,170.722,43.796,158.369
C06063=1034.082,249.204,-114.196,170.726,43.797,158.370
C06064=1034.091,249.546,-114.236,170.731,43.797,158.370
C06065=1034.098,249.795,-114.265,170.734,43.797,158.370
C06066=1034.104,250.043,-114.295,170.737,43.797,158.371
C06067=1034.110,250.290,-114.324,170.740,43.797,158.371
C06068=1034.117,250.539,-114.354,170.743,43.798,158.371
C06069=1034.124,250.787,-114.382,170.746,43.798,158.372
C06070=1034.130,251.035,-114.411,170.750,43.798,158.372
C06071=1034.137,251.284,-114.441,170.753,43.799,158.372
C06072=1034.144,251.532,-114.470,170.755,43.799,158.373
C06073=1034.150,251.779,-114.499,170.759,43.799,158.373
C06074=1034.157,252.028,-114.529,170.762,43.800,158.373
C06075=1034.164,252.276,-114.557,170.765,43.800,158.374
C06076=1034.171,252.525,-114.587,170.769,43.800,158.374
C06077=1034.177,252.772,-114.616,170.772,43.800,158.374
C06078=1034.184,253.021,-114.645,170.774,43.801,158.375
C06079=1034.190,253.269,-114.675,170.778,43.801,158.375
C06080=1034.197,253.518,-114.704,170.781,43.801,158.375
C06081=1034.205,253.765,-114.733,170.784,43.802,158.376
C06082=1034.211,254.014,-114.762,170.788,43.802,158.376
C06083=1034.217,254.262,-114.791,170.791,43.802,158.376
C06084=1034.224,254.510,-114.822,170.794,43.802,158.377
C06085=1034.230,254.758,-114.851,170.797,43.803,158.377
C06086=1034.237,255.007,-114.880,170.800,43.803,158.377
C06087=1034.245,255.254,-114.909,170.803,43.803,158.378
C06088=1034.251,255.503,-114.939,170.807,43.803,158.378
C06089=1034.258,255.751,-114.968,170.810,43.804,158.378
C06090=1034.265,255.999,-114.998,170.813,43.804,158.379
C06091=1034.271,256.247,-115.027,170.817,43.804,158.379
C06092=1034.278,256.496,-115.057,170.820,43.805,158.379
C06093=1034.285,256.744,-115.086,170.822,43.805,158.380
C06094=1034.291,256.993,-115.115,170.826,43.805,158.380
C06095=1034.299,257.240,-115.145,170.829,43.806,158.380
C06096=1034.306,257.489,-115.174,170.832,43.806,158.381
C06097=1034.312,257.736,-115.204,170.836,43.806,158.381
C06098=1034.319,257.985,-115.233,170.839,43.807,158.381
C06099=1034.325,258.232,-115.263,170.843,43.807,158.382
C06100=1034.332,258.481,-115.292,170.846,43.807,158.382
C06101=1034.339,258.729,-115.322,170.849,43.807,158.382
C06102=1034.346,258.977,-115.351,170.853,43.807,158.383
C06103=1034.354,259.226,-115.381,170.856,43.808,158.383
C06104=1034.360,259.474,-115.410,170.859,43.808,158.383
C06105=1034.367,259.722,-115.440,170.862,43.809,158.384
C06106=1034.374,259.969,-115.470,170.865,43.809,158.384
C06107=1034.380,260.218,-115.499,170.868,43.809,158.384
C06108=1034.388,260.466,-115.529,170.872,43.810,158.385
C06109=1034.394,260.715,-115.558,170.875,43.810,158.385
C06110=1034.402,260.963,-115.588,170.879,43.810,158.386
C06111=1034.408,261.210,-115.618,170.882,43.810,158.386
C06112=1034.415,261.459,-115.647,170.885,43.811,158.386
C06113=1034.422,261.707,-115.677,170.889,43.811,158.387
C06114=1034.428,261.955,-115.708,170.892,43.812,158.387
C06115=1034.435,262.203,-115.738,170.895,43.812,158.387
C06116=1034.442,262.451,-115.767,170.899,43.813,158.388
C06117=1034.451,262.791,-115.808,170.903,43.813,158.388
C06118=1034.460,263.131,-115.849,170.908,43.813,158.389
C06119=1034.469,263.471,-115.890,170.913,43.815,158.389
C06120=1034.478,263.811,-115.931,170.917,43.815,158.390
C06121=1034.485,264.059,-115.962,170.920,43.815,158.390
C06122=1034.491,264.307,-115.992,170.924,43.816,158.391
C06123=1034.498,264.555,-116.022,170.927,43.816,158.391
C06124=1034.506,264.803,-116.052,170.931,43.816,158.391
C06125=1034.511,265.051,-116.082,170.934,43.817,158.392
C06126=1034.519,265.299,-116.113,170.938,43.818,158.392
C06127=1034.526,265.547,-116.143,170.941,43.818,158.393
C06128=1034.532,265.795,-116.173,170.944,43.818,158.393
C06129=1034.538,266.044,-116.202,170.948,43.819,158.393
C06130=1034.546,266.292,-116.233,170.951,43.819,158.394
C06131=1034.552,266.540,-116.262,170.955,43.820,158.394
C06132=1034.559,266.788,-116.293,170.958,43.820,158.394
C06133=1034.566,267.036,-116.324,170.961,43.821,158.395
C06134=1034.573,267.283,-116.354,170.965,43.821,158.395
C06135=1034.579,267.532,-116.384,170.968,43.822,158.396
C06136=1034.586,267.780,-116.414,170.972,43.822,158.396
C06137=1034.592,268.028,-116.445,170.975,43.823,158.396
C06138=1034.599,268.276,-116.475,170.978,43.823,158.397
C06139=1034.605,268.525,-116.506,170.982,43.824,158.397
C06140=1034.613,268.773,-116.536,170.985,43.824,158.398
C06141=1034.620,269.020,-116.566,170.989,43.825,158.398
C06142=1034.626,269.268,-116.597,170.992,43.825,158.399
C06143=1034.633,269.517,-116.627,170.996,43.826,158.399
C06144=1034.640,269.765,-116.658,170.999,43.826,158.399
C06145=1034.646,270.013,-116.688,171.002,43.827,158.400
C06146=1034.653,270.261,-116.719,171.006,43.827,158.400
C06147=1034.660,270.509,-116.749,171.009,43.828,158.401
C06148=1034.666,270.757,-116.780,171.013,43.829,158.401
C06149=1034.673,271.005,-116.810,171.016,43.829,158.401
C06150=1034.680,271.253,-116.841,171.020,43.829,158.402
C06151=1034.687,271.501,-116.871,171.023,43.830,158.402
C06152=1034.693,271.749,-116.902,171.027,43.831,158.403
C06153=1034.700,271.996,-116.932,171.030,43.831,158.403
C06154=1034.707,272.245,-116.963,171.034,43.832,158.404
C06155=1034.713,272.493,-116.994,171.037,43.833,158.404
C06156=1034.720,272.741,-117.025,171.041,43.833,158.404
C06157=1034.727,272.989,-117.055,171.044,43.833,158.405
C06158=1034.734,273.236,-117.086,171.047,43.834,158.405
C06159=1034.740,273.485,-117.117,171.051,43.835,158.406
C06160=1034.747,273.733,-117.148,171.054,43.835,158.406
C06161=1034.754,273.981,-117.178,171.058,43.836,158.407
C06162=1034.761,274.229,-117.210,171.061,43.837,158.407
C06163=1034.767,274.477,-117.240,171.065,43.837,158.407
C06164=1034.774,274.724,-117.271,171.068,43.838,158.408
C06165=1034.780,274.973,-117.301,171.073,43.838,158.408
C06166=1034.787,275.221,-117.333,171.076,43.839,158.409
C06167=1034.794,275.469,-117.363,171.080,43.840,158.409
C06168=1034.801,275.717,-117.394,171.083,43.840,158.410
C06169=1034.807,275.965,-117.425,171.087,43.841,158.410
C06170=1034.815,276.213,-117.456,171.090,43.842,158.411
C06171=1034.822,276.461,-117.487,171.094,43.842,158.411
C06172=1034.827,276.709,-117.518,171.097,43.843,158.411
C06173=1034.838,277.053,-117.561,171.102,43.843,158.412
C06174=1034.847,277.398,-117.604,171.108,43.844,158.413
C06175=1034.856,277.742,-117.647,171.112,43.845,158.413
C06176=1034.865,278.087,-117.690,171.117,43.846,158.414
C06177=1034.873,278.335,-117.721,171.122,43.847,158.414
C06178=1034.879,278.583,-117.753,171.125,43.848,158.415
C06179=1034.886,278.831,-117.784,171.129,43.848,158.415
C06180=1034.892,279.079,-117.815,171.132,43.849,158.416
C06181=1034.899,279.327,-117.846,171.136,43.850,158.416
C06182=1034.906,279.575,-117.878,171.139,43.851,158.417
C06183=1034.913,279.823,-117.909,171.143,43.852,158.417
C06184=1034.919,280.071,-117.940,171.146,43.852,158.418
C06185=1034.926,280.319,-117.972,171.150,43.853,158.418
C06186=1034.933,280.567,-118.003,171.154,43.853,158.419
C06187=1034.940,280.814,-118.035,171.158,43.854,158.419
C06188=1034.946,281.063,-118.065,171.161,43.855,158.420
C06189=1034.953,281.311,-118.097,171.165,43.856,158.420
C06190=1034.959,281.559,-118.128,171.168,43.856,158.421
C06191=1034.966,281.807,-118.160,171.172,43.857,158.421
C06192=1034.973,282.055,-118.191,171.175,43.858,158.421
C06193=1034.980,282.302,-118.223,171.180,43.859,158.422
C06194=1034.987,282.550,-118.253,171.184,43.860,158.423
C06195=1034.994,282.798,-118.285,171.187,43.860,158.423
C06196=1035.000,283.046,-118.316,171.191,43.861,158.423
C06197=1035.007,283.294,-118.348,171.194,43.861,158.424
C06198=1035.014,283.542,-118.379,171.199,43.863,158.425
C06199=1035.021,283.790,-118.411,171.202,43.863,158.425
C06200=1035.028,284.037,-118.443,171.206,43.864,158.425
C06201=1035.034,284.285,-118.474,171.209,43.865,158.426
C06202=1035.041,284.533,-118.506,171.213,43.866,158.426
C06203=1035.048,284.781,-118.537,171.218,43.866,158.427
C06204=1035.055,285.028,-118.568,171.221,43.867,158.427
C06205=1035.061,285.276,-118.600,171.225,43.868,158.428
C06206=1035.069,285.525,-118.632,171.228,43.869,158.428
C06207=1035.076,285.772,-118.664,171.232,43.869,158.429
C06208=1035.082,286.020,-118.695,171.236,43.870,158.429
C06209=1035.089,286.268,-118.727,171.240,43.871,158.430
C06210=1035.096,286.516,-118.758,171.243,43.872,158.430
C06211=1035.103,286.764,-118.790,171.247,43.872,158.431
C06212=1035.110,287.011,-118.822,171.251,43.874,158.432
C06213=1035.116,287.259,-118.854,171.255,43.874,158.432
C06214=1035.123,287.508,-118.886,171.259,43.875,158.432
C06215=1035.130,287.755,-118.918,171.262,43.876,158.433
C06216=1035.137,288.003,-118.949,171.266,43.877,158.433
C06217=1035.143,288.251,-118.981,171.271,43.878,158.434
C06218=1035.150,288.498,-119.013,171.274,43.878,158.435
C06219=1035.156,288.747,-119.045,171.278,43.879,158.435
C06220=1035.164,288.995,-119.077,171.281,43.880,158.436
C06221=1035.171,289.242,-119.109,171.286,43.881,158.436
C06222=1035.178,289.490,-119.141,171.290,43.882,158.437
C06223=1035.184,289.738,-119.173,171.293,43.883,158.437
C06224=1035.191,289.985,-119.205,171.297,43.884,158.438
C06225=1035.198,290.234,-119.237,171.301,43.884,158.438
C06226=1035.205,290.481,-119.269,171.305,43.886,158.439
C06227=1035.211,290.729,-119.301,171.309,43.886,158.439
C06228=1035.218,290.977,-119.333,171.312,43.888,158.440
C06229=1035.228,291.334,-119.379,171.318,43.888,158.441
C06230=1035.239,291.691,-119.425,171.324,43.890,158.441
C06231=1035.248,292.046,-119.472,171.330,43.891,158.442
C06232=1035.258,292.403,-119.518,171.335,43.892,158.443
C06233=1035.265,292.651,-119.550,171.339,43.894,158.444
C06234=1035.271,292.900,-119.582,171.343,43.894,158.444
C06235=1035.279,293.147,-119.614,171.347,43.895,158.445
C06236=1035.286,293.394,-119.647,171.351,43.897,158.445
C06237=1035.292,293.642,-119.679,171.355,43.897,158.446
C06238=1035.299,293.890,-119.711,171.359,43.898,158.446
C06239=1035.305,294.138,-119.744,171.363,43.899,158.447
C06240=1035.312,294.385,-119.776,171.367,43.900,158.447
C06241=1035.320,294.633,-119.809,171.371,43.901,158.448
C06242=1035.326,294.881,-119.841,171.375,43.902,158.449
C06243=1035.333,295.129,-119.873,171.379,43.903,158.449
C06244=1035.340,295.377,-119.906,171.383,43.904,158.450
C06245=1035.346,295.625,-119.939,171.386,43.906,158.450
C06246=1035.353,295.872,-119.971,171.391,43.907,158.451
C06247=1035.360,296.119,-120.003,171.395,43.907,158.451
C06248=1035.367,296.368,-120.037,171.398,43.909,158.452
C06249=1035.373,296.615,-120.069,171.403,43.910,158.453
C06250=1035.380,296.863,-120.101,171.407,43.911,158.453
C06251=1035.387,297.111,-120.135,171.410,43.912,158.454
C06252=1035.393,297.359,-120.167,171.415,43.913,158.455
C06253=1035.400,297.606,-120.201,171.419,43.914,158.455
C06254=1035.407,297.853,-120.233,171.422,43.915,158.456
C06255=1035.414,298.101,-120.266,171.427,43.916,158.456
C06256=1035.420,298.349,-120.299,171.431,43.917,158.457
C06257=1035.427,298.597,-120.332,171.435,43.919,158.457
C06258=1035.434,298.844,-120.364,171.439,43.920,158.458
C06259=1035.441,299.093,-120.397,171.443,43.921,158.459
C06260=1035.447,299.340,-120.430,171.447,43.922,158.459
C06261=1035.454,299.588,-120.464,171.452,43.923,158.460
C06262=1035.461,299.835,-120.496,171.455,43.924,158.461
C06263=1035.468,300.083,-120.529,171.460,43.926,158.461
C06264=1035.474,300.331,-120.562,171.464,43.926,158.462
C06265=1035.481,300.578,-120.595,171.467,43.927,158.462
C06266=1035.489,300.826,-120.628,171.472,43.928,158.463
C06267=1035.495,301.074,-120.660,171.476,43.930,158.464
C06268=1035.502,301.322,-120.694,171.480,43.931,158.464
C06269=1035.508,301.569,-120.727,171.484,43.932,158.465
C06270=1035.516,301.817,-120.760,171.488,43.933,158.465
C06271=1035.522,302.064,-120.792,171.493,43.934,158.466
C06272=1035.530,302.312,-120.826,171.496,43.936,158.467
C06273=1035.536,302.560,-120.859,171.501,43.937,158.467
C06274=1035.543,302.808,-120.891,171.505,43.938,158.468
C06275=1035.551,303.055,-120.925,171.510,43.939,158.469
C06276=1035.557,303.303,-120.958,171.513,43.940,158.469
C06277=1035.564,303.551,-120.992,171.517,43.941,158.470
C06278=1035.570,303.798,-121.024,171.522,43.942,158.470
C06279=1035.578,304.046,-121.058,171.526,43.944,158.471
C06280=1035.585,304.293,-121.090,171.531,43.945,158.472
C06281=1035.592,304.541,-121.124,171.534,43.947,158.472
C06282=1035.599,304.789,-121.157,171.539,43.948,158.473
C06283=1035.606,305.036,-121.190,171.543,43.949,158.474
C06284=1035.613,305.284,-121.223,171.547,43.950,158.474
C06285=1035.623,305.657,-121.273,171.554,43.952,158.475
C06286=1035.634,306.031,-121.324,171.560,43.953,158.476
C06287=1035.644,306.404,-121.374,171.567,43.955,158.477
C06288=1035.655,306.778,-121.424,171.573,43.957,158.478
C06289=1035.662,307.026,-121.458,171.577,43.959,158.479
C06290=1035.669,307.273,-121.491,171.582,43.960,158.480
C06291=1035.676,307.521,-121.524,171.585,43.961,158.480
C06292=1035.684,307.768,-121.558,171.590,43.962,158.481
C06293=1035.690,308.015,-121.591,171.594,43.964,158.482
C06294=1035.697,308.263,-121.625,171.599,43.965,158.482
C06295=1035.704,308.511,-121.658,171.603,43.966,158.483
C06296=1035.712,308.759,-121.691,171.607,43.967,158.484
C06297=1035.719,309.006,-121.725,171.612,43.968,158.484
C06298=1035.726,309.253,-121.758,171.616,43.970,158.485
C06299=1035.733,309.502,-121.792,171.621,43.971,158.486
C06300=1035.740,309.749,-121.825,171.624,43.972,158.486
C06301=1035.748,309.997,-121.859,171.629,43.973,158.487
C06302=1035.755,310.244,-121.892,171.634,43.975,158.488
C06303=1035.762,310.491,-121.926,171.638,43.976,158.488
C06304=1035.769,310.739,-121.960,171.643,43.977,158.489
C06305=1035.776,310.987,-121.993,171.646,43.978,158.490
C06306=1035.783,311.235,-122.027,171.651,43.980,158.490
C06307=1035.791,311.482,-122.060,171.656,43.981,158.491
C06308=1035.798,311.730,-122.094,171.660,43.982,158.492
C06309=1035.804,311.977,-122.128,171.665,43.984,158.492
C06310=1035.811,312.225,-122.162,171.669,43.985,158.493
C06311=1035.819,312.472,-122.196,171.673,43.987,158.494
C06312=1035.825,312.720,-122.231,171.677,43.989,158.495
C06313=1035.833,312.968,-122.264,171.682,43.990,158.495
C06314=1035.838,313.215,-122.298,171.686,43.992,158.496
C06315=1035.846,313.462,-122.332,171.691,43.993,158.497
C06316=1035.853,313.710,-122.367,171.696,43.994,158.498
C06317=1035.860,313.958,-122.401,171.700,43.996,158.498
C06318=1035.867,314.205,-122.435,171.705,43.997,158.499
C06319=1035.873,314.453,-122.469,171.709,43.999,158.500
C06320=1035.880,314.700,-122.504,171.713,44.000,158.500
C06321=1035.887,314.948,-122.538,171.718,44.002,158.501
C06322=1035.894,315.195,-122.572,171.722,44.003,158.502
C06323=1035.901,315.442,-122.606,171.727,44.005,158.503
C06324=1035.908,315.690,-122.641,171.731,44.006,158.503
C06325=1035.915,315.937,-122.675,171.736,44.008,158.504
C06326=1035.922,316.185,-122.710,171.741,44.009,158.505
C06327=1035.929,316.433,-122.744,171.745,44.011,158.506
C06328=1035.936,316.680,-122.779,171.750,44.012,158.506
C06329=1035.943,316.928,-122.813,171.754,44.014,158.507
C06330=1035.950,317.175,-122.847,171.758,44.015,158.508
C06331=1035.957,317.423,-122.882,171.763,44.017,158.509
C06332=1035.964,317.670,-122.916,171.767,44.019,158.509
C06333=1035.971,317.918,-122.951,171.772,44.020,158.510
C06334=1035.978,318.165,-122.985,171.777,44.021,158.511
C06335=1035.985,318.413,-123.019,171.781,44.023,158.512
C06336=1035.992,318.660,-123.054,171.786,44.025,158.512
C06337=1035.999,318.908,-123.088,171.791,44.027,158.513
C06338=1036.006,319.155,-123.123,171.795,44.028,158.514
C06339=1036.013,319.403,-123.158,171.800,44.029,158.515
C06340=1036.020,319.650,-123.192,171.805,44.031,158.516
C06341=1036.031,320.028,-123.245,171.811,44.034,158.517
C06342=1036.042,320.406,-123.298,171.819,44.036,158.518
C06343=1036.053,320.784,-123.350,171.826,44.039,158.519
C06344=1036.065,321.163,-123.404,171.834,44.041,158.520
C06345=1036.071,321.410,-123.439,171.838,44.043,158.521
C06346=1036.079,321.658,-123.473,171.843,44.044,158.522
C06347=1036.085,321.905,-123.508,171.848,44.046,158.523
C06348=1036.093,322.152,-123.543,171.853,44.048,158.524
C06349=1036.100,322.400,-123.578,171.857,44.050,158.524
C06350=1036.108,322.648,-123.613,171.862,44.051,158.525
C06351=1036.114,322.896,-123.647,171.867,44.053,158.526
C06352=1036.122,323.143,-123.682,171.871,44.054,158.527
C06353=1036.128,323.390,-123.717,171.875,44.056,158.528
C06354=1036.137,323.638,-123.752,171.880,44.058,158.528
C06355=1036.143,323.885,-123.787,171.885,44.059,158.529
C06356=1036.151,324.132,-123.821,171.890,44.061,158.530
C06357=1036.158,324.380,-123.856,171.895,44.063,158.531
C06358=1036.166,324.627,-123.891,171.899,44.065,158.532
C06359=1036.172,324.875,-123.926,171.904,44.066,158.532
C06360=1036.180,325.122,-123.961,171.909,44.068,158.533
C06361=1036.187,325.370,-123.996,171.914,44.069,158.534
C06362=1036.195,325.617,-124.031,171.919,44.071,158.535
C06363=1036.202,325.864,-124.066,171.923,44.073,158.536
C06364=1036.210,326.112,-124.101,171.928,44.074,158.537
C06365=1036.216,326.359,-124.136,171.933,44.076,158.537
C06366=1036.225,326.607,-124.171,171.938,44.078,158.538
C06367=1036.231,326.854,-124.206,171.944,44.080,158.539
C06368=1036.239,327.101,-124.241,171.948,44.082,158.540
C06369=1036.246,327.350,-124.276,171.953,44.083,158.541
C06370=1036.254,327.596,-124.312,171.957,44.085,158.542
C06371=1036.261,327.844,-124.347,171.962,44.087,158.542
C06372=1036.269,328.091,-124.382,171.967,44.088,158.543
C06373=1036.276,328.339,-124.417,171.973,44.090,158.544
C06374=1036.283,328.587,-124.452,171.978,44.092,158.545
C06375=1036.290,328.833,-124.488,171.983,44.094,158.546
C06376=1036.297,329.081,-124.524,171.988,44.096,158.547
C06377=1036.305,329.328,-124.559,171.992,44.098,158.548
C06378=1036.313,329.576,-124.594,171.997,44.100,158.549
C06379=1036.320,329.823,-124.630,172.002,44.101,158.549
C06380=1036.327,330.071,-124.666,172.007,44.104,158.550
C06381=1036.334,330.318,-124.701,172.012,44.105,158.551
C06382=1036.341,330.565,-124.737,172.017,44.107,158.552
C06383=1036.349,330.812,-124.773,172.023,44.109,158.553
C06384=1036.355,331.060,-124.808,172.028,44.111,158.554
C06385=1036.363,331.307,-124.844,172.033,44.113,158.555
C06386=1036.370,331.554,-124.879,172.037,44.115,158.556
C06387=1036.378,331.802,-124.916,172.042,44.117,158.557
C06388=1036.384,332.049,-124.951,172.047,44.119,158.558
C06389=1036.392,332.297,-124.987,172.052,44.121,158.558
C06390=1036.400,332.544,-125.023,172.057,44.123,158.559
C06391=1036.406,332.791,-125.058,172.062,44.125,158.560
C06392=1036.414,333.039,-125.094,172.068,44.127,158.561
C06393=1036.421,333.286,-125.130,172.073,44.128,158.562
C06394=1036.429,333.533,-125.167,172.078,44.131,158.563
C06395=1036.436,333.781,-125.202,172.083,44.133,158.564
C06396=1036.443,334.028,-125.238,172.088,44.134,158.565
C06397=1036.452,334.328,-125.282,172.095,44.137,158.566
C06398=1036.461,334.628,-125.325,172.101,44.140,158.567
C06399=1036.470,334.928,-125.369,172.106,44.142,158.568
C06400=1036.480,335.228,-125.413,172.113,44.144,158.569
C06401=1036.487,335.476,-125.449,172.118,44.147,158.570
C06402=1036.494,335.723,-125.485,172.123,44.149,158.571
C06403=1036.501,335.970,-125.521,172.128,44.151,158.572
C06404=1036.509,336.217,-125.558,172.134,44.153,158.573
C06405=1036.516,336.464,-125.593,172.139,44.155,158.574
C06406=1036.524,336.712,-125.630,172.144,44.157,158.575
C06407=1036.531,336.959,-125.666,172.149,44.159,158.576
C06408=1036.538,337.206,-125.702,172.154,44.161,158.577
C06409=1036.545,337.454,-125.739,172.160,44.163,158.578
C06410=1036.553,337.701,-125.775,172.165,44.166,158.579
C06411=1036.561,337.948,-125.811,172.170,44.168,158.580
C06412=1036.567,338.195,-125.848,172.175,44.170,158.581
C06413=1036.575,338.442,-125.884,172.181,44.172,158.582
C06414=1036.583,338.690,-125.921,172.186,44.174,158.583
C06415=1036.590,338.937,-125.957,172.191,44.177,158.584
C06416=1036.597,339.185,-125.994,172.196,44.179,158.585
C06417=1036.605,339.431,-126.030,172.203,44.181,158.586
C06418=1036.612,339.679,-126.066,172.208,44.183,158.587
C06419=1036.620,339.926,-126.103,172.213,44.185,158.588
C06420=1036.627,340.174,-126.139,172.218,44.187,158.589
C06421=1036.635,340.421,-126.176,172.224,44.190,158.590
C06422=1036.643,340.668,-126.213,172.229,44.192,158.591
C06423=1036.651,340.915,-126.250,172.234,44.194,158.592
C06424=1036.657,341.162,-126.286,172.239,44.196,158.593
C06425=1036.667,341.483,-126.334,172.247,44.199,158.594
C06426=1036.676,341.803,-126.382,172.254,44.202,158.596
C06427=1036.687,342.124,-126.429,172.260,44.205,158.597
C06428=1036.696,342.444,-126.477,172.268,44.208,158.598
C06429=1036.703,342.692,-126.513,172.273,44.211,158.599
C06430=1036.711,342.939,-126.551,172.279,44.213,158.600
C06431=1036.718,343.186,-126.587,172.284,44.215,158.601
C06432=1036.726,343.433,-126.625,172.289,44.218,158.603
C06433=1036.733,343.680,-126.662,172.295,44.220,158.604
C06434=1036.740,343.928,-126.698,172.300,44.222,158.605
C06435=1036.748,344.175,-126.735,172.306,44.225,158.606
C06436=1036.756,344.422,-126.773,172.312,44.227,158.607
C06437=1036.764,344.669,-126.810,172.317,44.229,158.608
C06438=1036.771,344.917,-126.847,172.322,44.232,158.609
C06439=1036.779,345.163,-126.883,172.328,44.234,158.610
C06440=1036.786,345.411,-126.921,172.334,44.236,158.611
C06441=1036.794,345.657,-126.958,172.339,44.239,158.612
C06442=1036.801,345.904,-126.995,172.345,44.241,158.613
C06443=1036.809,346.151,-127.032,172.350,44.244,158.614
C06444=1036.816,346.398,-127.070,172.356,44.246,158.615
C06445=1036.824,346.646,-127.108,172.362,44.248,158.616
C06446=1036.832,346.893,-127.145,172.367,44.251,158.618
C06447=1036.839,347.140,-127.182,172.373,44.254,158.619
C06448=1036.847,347.387,-127.219,172.378,44.256,158.620
C06449=1036.855,347.634,-127.257,172.385,44.258,158.621
C06450=1036.862,347.881,-127.294,172.390,44.261,158.622
C06451=1036.870,348.128,-127.331,172.395,44.263,158.623
C06452=1036.878,348.376,-127.369,172.401,44.266,158.624
C06453=1036.889,348.747,-127.425,172.410,44.269,158.626
C06454=1036.901,349.115,-127.481,172.418,44.274,158.628
C06455=1036.912,349.486,-127.537,172.427,44.277,158.629
C06456=1036.923,349.856,-127.594,172.435,44.281,158.631
C06457=1036.931,350.104,-127.631,172.441,44.284,158.632
C06458=1036.938,350.351,-127.669,172.447,44.286,158.633
C06459=1036.946,350.597,-127.707,172.453,44.289,158.635
C06460=1036.954,350.844,-127.744,172.458,44.292,158.636
C06461=1036.962,351.091,-127.783,172.465,44.294,158.637
C06462=1036.969,351.339,-127.820,172.470,44.297,158.638
C06463=1036.977,351.586,-127.858,172.476,44.299,158.639
C06464=1036.984,351.832,-127.896,172.482,44.302,158.640
C06465=1036.992,352.080,-127.934,172.488,44.305,158.641
C06466=1037.000,352.327,-127.972,172.493,44.307,158.643
C06467=1037.007,352.573,-128.009,172.500,44.310,158.644
C06468=1037.016,352.821,-128.048,172.505,44.313,158.645
C06469=1037.023,353.068,-128.085,172.511,44.316,158.646
C06470=1037.030,353.314,-128.123,172.517,44.318,158.648
C06471=1037.039,353.561,-128.162,172.523,44.321,158.649
C06472=1037.046,353.809,-128.200,172.529,44.324,158.650
C06473=1037.054,354.056,-128.238,172.535,44.326,158.651
C06474=1037.062,354.302,-128.276,172.540,44.329,158.652
C06475=1037.070,354.549,-128.313,172.547,44.332,158.653
C06476=1037.078,354.796,-128.352,172.552,44.334,158.655
C06477=1037.085,355.043,-128.390,172.559,44.338,158.656
C06478=1037.093,355.290,-128.429,172.565,44.340,158.657
C06479=1037.101,355.537,-128.466,172.571,44.343,158.658
C06480=1037.109,355.784,-128.505,172.577,44.346,158.659
C06481=1037.116,356.031,-128.543,172.582,44.349,158.661
C06482=1037.124,356.278,-128.582,172.589,44.351,158.662
C06483=1037.132,356.525,-128.620,172.594,44.354,158.663
C06484=1037.140,356.772,-128.659,172.601,44.357,158.665
C06485=1037.148,357.018,-128.697,172.607,44.360,158.666
C06486=1037.156,357.266,-128.736,172.613,44.363,158.667
C06487=1037.163,357.512,-128.774,172.619,44.366,158.668
C06488=1037.172,357.759,-128.812,172.626,44.368,158.670
C06489=1037.179,358.006,-128.851,172.631,44.372,158.671
C06490=1037.187,358.253,-128.889,172.638,44.374,158.672
C06491=1037.195,358.500,-128.928,172.644,44.378,158.673
C06492=1037.203,358.747,-128.966,172.650,44.380,158.675
C06493=1037.211,358.994,-129.005,172.656,44.383,158.676
C06494=1037.219,359.241,-129.045,172.662,44.386,158.677
C06495=1037.226,359.488,-129.083,172.668,44.389,158.679
C06496=1037.235,359.735,-129.121,172.675,44.392,158.680
C06497=1037.242,359.981,-129.160,172.681,44.395,158.681
C06498=1037.251,360.228,-129.199,172.687,44.398,158.682
C06499=1037.259,360.475,-129.238,172.694,44.401,158.684
C06500=1037.267,360.722,-129.276,172.699,44.404,158.685
C06501=1037.274,360.968,-129.316,172.706,44.407,158.686
C06502=1037.282,361.216,-129.354,172.712,44.410,158.688
C06503=1037.291,361.462,-129.394,172.719,44.413,158.689
C06504=1037.298,361.709,-129.432,172.725,44.416,158.690
C06505=1037.306,361.956,-129.471,172.731,44.419,158.692
C06506=1037.314,362.203,-129.511,172.738,44.422,158.693
C06507=1037.322,362.450,-129.550,172.745,44.425,158.694
C06508=1037.329,362.696,-129.589,172.750,44.429,158.696
C06509=1037.342,363.072,-129.649,172.760,44.433,158.698
C06510=1037.354,363.448,-129.708,172.770,44.438,158.700
C06511=1037.366,363.825,-129.769,172.780,44.443,158.702
C06512=1037.378,364.201,-129.828,172.789,44.448,158.704
C06513=1037.386,364.448,-129.868,172.796,44.451,158.706
C06514=1037.395,364.694,-129.907,172.803,44.454,158.707
C06515=1037.402,364.941,-129.947,172.810,44.457,158.708
C06516=1037.411,365.188,-129.986,172.815,44.461,158.710
C06517=1037.419,365.435,-130.025,172.822,44.464,158.711
C06518=1037.427,365.682,-130.065,172.829,44.467,158.712
C06519=1037.434,365.928,-130.104,172.835,44.470,158.714
C06520=1037.442,366.175,-130.144,172.842,44.474,158.715
C06521=1037.451,366.421,-130.183,172.849,44.477,158.717
C06522=1037.458,366.668,-130.223,172.855,44.480,158.718
C06523=1037.467,366.915,-130.262,172.861,44.483,158.719
C06524=1037.475,367.162,-130.302,172.868,44.487,158.721
C06525=1037.483,367.408,-130.341,172.875,44.490,158.722
C06526=1037.492,367.654,-130.382,172.882,44.493,158.724
C06527=1037.499,367.901,-130.421,172.888,44.497,158.725
C06528=1037.508,368.148,-130.461,172.895,44.500,158.727
C06529=1037.516,368.396,-130.501,172.902,44.503,158.728
C06530=1037.525,368.642,-130.540,172.908,44.506,158.730
C06531=1037.532,368.889,-130.580,172.915,44.510,158.731
C06532=1037.541,369.135,-130.620,172.922,44.513,158.733
C06533=1037.550,369.382,-130.660,172.928,44.516,158.734
C06534=1037.557,369.629,-130.700,172.935,44.520,158.736
C06535=1037.566,369.874,-130.740,172.942,44.523,158.737
C06536=1037.574,370.122,-130.780,172.949,44.527,158.739
C06537=1037.582,370.369,-130.820,172.956,44.530,158.740
C06538=1037.591,370.615,-130.860,172.963,44.533,158.741
C06539=1037.599,370.862,-130.900,172.970,44.537,158.743
C06540=1037.607,371.108,-130.940,172.976,44.541,158.745
C06541=1037.615,371.354,-130.981,172.983,44.545,158.746
C06542=1037.623,371.601,-131.020,172.990,44.548,158.748
C06543=1037.632,371.848,-131.061,172.997,44.551,158.749
C06544=1037.640,372.095,-131.101,173.004,44.555,158.751
C06545=1037.648,372.341,-131.142,173.011,44.558,158.752
C06546=1037.656,372.588,-131.183,173.018,44.562,158.754
C06547=1037.664,372.833,-131.223,173.025,44.566,158.755
C06548=1037.673,373.081,-131.263,173.032,44.569,158.757
C06549=1037.681,373.327,-131.304,173.039,44.573,158.758
C06550=1037.689,373.574,-131.344,173.046,44.577,158.760
C06551=1037.697,373.821,-131.385,173.053,44.580,158.762
C06552=1037.706,374.067,-131.425,173.060,44.584,158.763
C06553=1037.714,374.313,-131.466,173.067,44.587,158.765
C06554=1037.723,374.560,-131.507,173.074,44.591,158.766
C06555=1037.731,374.806,-131.547,173.081,44.595,158.768
C06556=1037.740,375.052,-131.587,173.088,44.598,158.769
C06557=1037.748,375.299,-131.628,173.095,44.602,158.771
C06558=1037.756,375.545,-131.669,173.103,44.605,158.773
C06559=1037.765,375.792,-131.710,173.110,44.610,158.774
C06560=1037.773,376.039,-131.751,173.117,44.613,158.776
C06561=1037.782,376.285,-131.791,173.124,44.617,158.778
C06562=1037.790,376.532,-131.832,173.131,44.620,158.779
C06563=1037.799,376.779,-131.873,173.138,44.625,158.781
C06564=1037.807,377.025,-131.913,173.145,44.628,158.782
C06565=1037.821,377.421,-131.980,173.157,44.634,158.785
C06566=1037.835,377.818,-132.045,173.169,44.640,158.788
C06567=1037.849,378.214,-132.111,173.181,44.647,158.790
C06568=1037.862,378.611,-132.178,173.192,44.653,158.793
C06569=1037.870,378.857,-132.218,173.200,44.657,158.795
C06570=1037.879,379.104,-132.260,173.207,44.660,158.796
C06571=1037.887,379.350,-132.301,173.214,44.665,158.798
C06572=1037.896,379.596,-132.342,173.222,44.668,158.800
C06573=1037.904,379.842,-132.384,173.230,44.673,158.802
C06574=1037.913,380.089,-132.425,173.237,44.676,158.803
C06575=1037.921,380.336,-132.467,173.244,44.680,158.805
C06576=1037.930,380.581,-132.509,173.252,44.685,158.807
C06577=1037.938,380.828,-132.550,173.260,44.688,158.809
C06578=1037.947,381.075,-132.591,173.267,44.693,158.810
C06579=1037.956,381.320,-132.633,173.274,44.696,158.812
C06580=1037.964,381.567,-132.675,173.282,44.700,158.814
C06581=1037.972,381.814,-132.716,173.289,44.704,158.815
C06582=1037.981,382.060,-132.758,173.297,44.708,158.817
C06583=1037.990,382.306,-132.799,173.305,44.713,158.819
C06584=1037.999,382.552,-132.841,173.312,44.717,158.821
C06585=1038.008,382.799,-132.882,173.320,44.721,158.822
C06586=1038.016,383.045,-132.925,173.328,44.725,158.824
C06587=1038.025,383.292,-132.966,173.335,44.729,158.826
C06588=1038.033,383.537,-133.008,173.343,44.733,158.828
C06589=1038.042,383.784,-133.049,173.351,44.738,158.830
C06590=1038.051,384.030,-133.091,173.358,44.742,158.831
C06591=1038.060,384.276,-133.133,173.367,44.746,158.833
C06592=1038.068,384.522,-133.176,173.374,44.750,158.835
C06593=1038.077,384.769,-133.218,173.381,44.754,158.837
C06594=1038.086,385.015,-133.259,173.390,44.758,158.839
C06595=1038.095,385.262,-133.301,173.397,44.762,158.841
C06596=1038.104,385.507,-133.344,173.406,44.766,158.842
C06597=1038.113,385.754,-133.386,173.413,44.771,158.844
C06598=1038.122,386.000,-133.428,173.421,44.775,158.846
C06599=1038.131,386.246,-133.470,173.429,44.779,158.848
C06600=1038.140,386.492,-133.512,173.437,44.784,158.850
C06601=1038.149,386.739,-133.553,173.445,44.788,158.852
C06602=1038.157,386.985,-133.596,173.453,44.792,158.854
C06603=1038.166,387.231,-133.638,173.461,44.796,158.855
C06604=1038.175,387.477,-133.681,173.469,44.801,158.857
C06605=1038.184,387.723,-133.722,173.477,44.805,158.859
C06606=1038.193,387.969,-133.765,173.485,44.809,158.861
C06607=1038.203,388.216,-133.808,173.493,44.814,158.863
C06608=1038.212,388.462,-133.850,173.501,44.819,158.865
C06609=1038.220,388.708,-133.893,173.509,44.823,158.867
C06610=1038.229,388.954,-133.935,173.517,44.827,158.869
C06611=1038.238,389.200,-133.978,173.525,44.832,158.871
C06612=1038.247,389.446,-134.021,173.533,44.836,158.873
C06613=1038.255,389.692,-134.063,173.542,44.841,158.875
C06614=1038.265,389.939,-134.106,173.550,44.845,158.877
C06615=1038.274,390.185,-134.149,173.558,44.850,158.879
C06616=1038.283,390.431,-134.191,173.567,44.854,158.881
C06617=1038.291,390.677,-134.234,173.574,44.859,158.883
C06618=1038.301,390.923,-134.277,173.583,44.863,158.885
C06619=1038.310,391.169,-134.320,173.591,44.868,158.886
C06620=1038.319,391.415,-134.363,173.599,44.872,158.888
C06621=1038.327,391.630,-134.401,173.606,44.877,158.890
C06622=1038.335,391.846,-134.438,173.614,44.881,158.892
C06623=1038.343,392.061,-134.476,173.621,44.885,158.894
C06624=1038.350,392.277,-134.514,173.629,44.889,158.896
C06625=1038.359,392.492,-134.552,173.636,44.893,158.897
C06626=1038.367,392.708,-134.590,173.643,44.897,158.899
C06627=1038.374,392.924,-134.628,173.651,44.901,158.901
C06628=1038.383,393.138,-134.666,173.658,44.906,158.903
C06629=1038.391,393.384,-134.709,173.667,44.910,158.905
C06630=1038.401,393.631,-134.751,173.676,44.914,158.907
C06631=1038.410,393.876,-134.795,173.684,44.920,158.909
C06632=1038.419,394.123,-134.838,173.692,44.924,158.911
C06633=1038.429,394.368,-134.882,173.701,44.929,158.913
C06634=1038.438,394.615,-134.925,173.710,44.934,158.915
C06635=1038.447,394.860,-134.969,173.719,44.938,158.917
C06636=1038.457,395.106,-135.012,173.727,44.944,158.919
C06637=1038.465,395.352,-135.055,173.736,44.949,158.922
C06638=1038.475,395.598,-135.099,173.744,44.953,158.924
C06639=1038.484,395.844,-135.144,173.753,44.958,158.926
C06640=1038.493,396.090,-135.187,173.762,44.963,158.928
C06641=1038.503,396.336,-135.230,173.771,44.968,158.930
C06642=1038.512,396.582,-135.274,173.779,44.973,158.932
C06643=1038.521,396.828,-135.318,173.788,44.978,158.934
C06644=1038.530,397.074,-135.362,173.797,44.983,158.937
C06645=1038.539,397.319,-135.406,173.806,44.988,158.939
C06646=1038.549,397.566,-135.450,173.815,44.993,158.941
C06647=1038.559,397.811,-135.493,173.824,44.998,158.943
C06648=1038.568,398.058,-135.537,173.833,45.003,158.945
C06649=1038.577,398.303,-135.581,173.842,45.008,158.948
C06650=1038.587,398.549,-135.626,173.850,45.013,158.950
C06651=1038.596,398.795,-135.670,173.860,45.018,158.952
C06652=1038.605,399.041,-135.714,173.869,45.023,158.954
C06653=1038.615,399.286,-135.757,173.878,45.028,158.957
C06654=1038.624,399.532,-135.802,173.887,45.034,158.959
C06655=1038.634,399.778,-135.846,173.896,45.038,158.961
C06656=1038.644,400.024,-135.890,173.905,45.043,158.963
C06657=1038.653,400.270,-135.935,173.914,45.049,158.966
C06658=1038.663,400.515,-135.979,173.923,45.054,158.968
C06659=1038.672,400.761,-136.023,173.932,45.059,158.970
C06660=1038.682,401.007,-136.068,173.941,45.064,158.972
C06661=1038.691,401.253,-136.112,173.951,45.069,158.975
C06662=1038.701,401.499,-136.157,173.960,45.075,158.977
C06663=1038.711,401.744,-136.202,173.969,45.080,158.979
C06664=1038.720,401.990,-136.246,173.979,45.085,158.982
C06665=1038.730,402.236,-136.291,173.988,45.091,158.984
C06666=1038.739,402.482,-136.336,173.997,45.096,158.986
C06667=1038.748,402.728,-136.381,174.007,45.101,158.989
C06668=1038.758,402.973,-136.425,174.017,45.107,158.991
C06669=1038.768,403.219,-136.470,174.026,45.112,158.994
C06670=1038.777,403.464,-136.515,174.035,45.118,158.996
C06671=1038.788,403.711,-136.560,174.044,45.123,158.998
C06672=1038.797,403.956,-136.606,174.055,45.129,159.001
C06673=1038.806,404.202,-136.650,174.064,45.134,159.003
C06674=1038.816,404.447,-136.695,174.073,45.139,159.006
C06675=1038.825,404.693,-136.741,174.082,45.145,159.008
C06676=1038.835,404.939,-136.786,174.093,45.151,159.011
C06677=1038.845,405.185,-136.831,174.102,45.156,159.013
C06678=1038.855,405.430,-136.876,174.111,45.162,159.015
C06679=1038.864,405.676,-136.922,174.122,45.167,159.018
C06680=1038.874,405.922,-136.967,174.131,45.173,159.020
C06681=1038.883,406.147,-137.008,174.140,45.178,159.023
C06682=1038.892,406.373,-137.050,174.149,45.183,159.025
C06683=1038.901,406.598,-137.092,174.159,45.188,159.027
C06684=1038.910,406.823,-137.134,174.168,45.193,159.030
C06685=1038.919,407.048,-137.175,174.177,45.199,159.032
C06686=1038.928,407.274,-137.217,174.185,45.204,159.034
C06687=1038.937,407.498,-137.259,174.194,45.209,159.037
C06688=1038.947,407.725,-137.301,174.203,45.215,159.039
C06689=1038.956,407.970,-137.346,174.214,45.220,159.041
C06690=1038.967,408.216,-137.392,174.223,45.226,159.044
C06691=1038.977,408.461,-137.438,174.234,45.231,159.047
C06692=1038.986,408.707,-137.483,174.243,45.237,159.049
C06693=1038.996,408.952,-137.529,174.254,45.243,159.052
C06694=1039.007,409.198,-137.575,174.264,45.249,159.054
C06695=1039.017,409.444,-137.621,174.274,45.255,159.057
C06696=1039.027,409.689,-137.667,174.284,45.261,159.060
C06697=1039.037,409.935,-137.712,174.294,45.266,159.062
C06698=1039.047,410.181,-137.758,174.305,45.272,159.065
C06699=1039.057,410.426,-137.804,174.315,45.278,159.067
C06700=1039.068,410.671,-137.850,174.325,45.284,159.070
C06701=1039.078,410.917,-137.896,174.336,45.290,159.073
C06702=1039.088,411.163,-137.942,174.346,45.296,159.075
C06703=1039.099,411.408,-137.988,174.357,45.302,159.078
C06704=1039.109,411.654,-138.035,174.367,45.308,159.081
C06705=1039.119,411.900,-138.082,174.377,45.314,159.083
C06706=1039.129,412.144,-138.127,174.388,45.320,159.086
C06707=1039.139,412.390,-138.174,174.399,45.326,159.089
C06708=1039.150,412.635,-138.221,174.408,45.332,159.092
C06709=1039.160,412.881,-138.267,174.419,45.338,159.094
C06710=1039.170,413.127,-138.314,174.430,45.345,159.097
C06711=1039.180,413.372,-138.360,174.441,45.351,159.100
C06712=1039.191,413.617,-138.407,174.452,45.357,159.103
C06713=1039.200,413.863,-138.454,174.463,45.363,159.106
C06714=1039.211,414.108,-138.501,174.472,45.369,159.108
C06715=1039.222,414.354,-138.548,174.483,45.375,159.111
C06716=1039.232,414.599,-138.595,174.494,45.382,159.114
C06717=1039.242,414.845,-138.641,174.505,45.388,159.117
C06718=1039.253,415.090,-138.688,174.516,45.394,159.120
C06719=1039.263,415.335,-138.735,174.527,45.401,159.123
C06720=1039.273,415.580,-138.783,174.538,45.407,159.125
C06721=1039.284,415.825,-138.829,174.549,45.413,159.128
C06722=1039.294,416.071,-138.876,174.560,45.420,159.131
C06723=1039.305,416.317,-138.924,174.571,45.426,159.134
C06724=1039.316,416.561,-138.971,174.582,45.433,159.137
C06725=1039.326,416.807,-139.018,174.593,45.439,159.140
C06726=1039.336,417.052,-139.065,174.605,45.445,159.143
C06727=1039.348,417.298,-139.112,174.616,45.452,159.146
C06728=1039.358,417.543,-139.159,174.627,45.458,159.149
C06729=1039.368,417.788,-139.207,174.638,45.464,159.152
C06730=1039.379,418.034,-139.255,174.649,45.471,159.155
C06731=1039.389,418.279,-139.302,174.660,45.478,159.158
C06732=1039.400,418.524,-139.350,174.672,45.484,159.161
C06733=1039.411,418.770,-139.397,174.684,45.491,159.164
C06734=1039.421,419.014,-139.445,174.695,45.498,159.167
C06735=1039.432,419.260,-139.493,174.706,45.504,159.170
C06736=1039.443,419.505,-139.540,174.718,45.511,159.173
C06737=1039.454,419.750,-139.589,174.729,45.517,159.176
C06738=1039.464,419.995,-139.636,174.741,45.525,159.179
C06739=1039.476,420.241,-139.684,174.753,45.531,159.182
C06740=1039.486,420.485,-139.732,174.764,45.538,159.185
C06741=1039.496,420.715,-139.777,174.776,45.544,159.188
C06742=1039.506,420.944,-139.823,174.786,45.551,159.191
C06743=1039.516,421.174,-139.868,174.797,45.557,159.194
C06744=1039.527,421.404,-139.912,174.809,45.563,159.197
C06745=1039.537,421.633,-139.958,174.820,45.570,159.200
C06746=1039.547,421.863,-140.003,174.831,45.576,159.203
C06747=1039.557,422.092,-140.048,174.842,45.583,159.206
C06748=1039.568,422.321,-140.093,174.853,45.589,159.209
C06749=1039.579,422.567,-140.141,174.865,45.596,159.212
C06750=1039.590,422.812,-140.189,174.877,45.603,159.215
C06751=1039.601,423.057,-140.238,174.889,45.610,159.219
C06752=1039.612,423.301,-140.286,174.901,45.617,159.222
C06753=1039.623,423.547,-140.335,174.913,45.624,159.225
C06754=1039.634,423.792,-140.384,174.926,45.631,159.228
C06755=1039.645,424.037,-140.432,174.938,45.638,159.232
C06756=1039.656,424.282,-140.482,174.950,45.645,159.235
C06757=1039.667,424.527,-140.530,174.963,45.652,159.238
C06758=1039.679,424.772,-140.579,174.975,45.659,159.242
C06759=1039.690,425.017,-140.628,174.987,45.666,159.245
C06760=1039.701,425.262,-140.676,175.000,45.674,159.248
C06761=1039.712,425.507,-140.726,175.012,45.681,159.252
C06762=1039.723,425.752,-140.775,175.025,45.688,159.255
C06763=1039.735,425.997,-140.824,175.038,45.695,159.259
C06764=1039.746,426.242,-140.873,175.051,45.703,159.262
C06765=1039.757,426.487,-140.922,175.062,45.710,159.265
C06766=1039.768,426.731,-140.971,175.075,45.717,159.269
C06767=1039.779,426.976,-141.020,175.088,45.724,159.272
C06768=1039.791,427.222,-141.070,175.101,45.732,159.276
C06769=1039.803,427.466,-141.119,175.113,45.739,159.279
C06770=1039.813,427.711,-141.168,175.126,45.747,159.283
C06771=1039.826,427.956,-141.219,175.139,45.754,159.286
C06772=1039.837,428.201,-141.268,175.152,45.762,159.290
C06773=1039.848,428.446,-141.317,175.165,45.769,159.293
C06774=1039.860,428.690,-141.367,175.179,45.776,159.297
C06775=1039.871,428.936,-141.417,175.192,45.784,159.301
C06776=1039.883,429.180,-141.467,175.205,45.792,159.304
C06777=1039.894,429.424,-141.517,175.218,45.800,159.308
C06778=1039.906,429.670,-141.566,175.231,45.807,159.311
C06779=1039.917,429.914,-141.617,175.244,45.815,159.315
C06780=1039.929,430.159,-141.667,175.258,45.822,159.318
C06781=1039.940,430.403,-141.717,175.271,45.830,159.322
C06782=1039.952,430.648,-141.767,175.284,45.838,159.326
C06783=1039.963,430.893,-141.817,175.299,45.845,159.330
C06784=1039.975,431.138,-141.868,175.312,45.853,159.333
C06785=1039.986,431.382,-141.918,175.325,45.861,159.337
C06786=1039.999,431.627,-141.968,175.339,45.869,159.341
C06787=1040.010,431.872,-142.019,175.352,45.876,159.344
C06788=1040.022,432.116,-142.068,175.367,45.884,159.348
C06789=1040.034,432.361,-142.118,175.380,45.892,159.352
C06790=1040.046,432.605,-142.170,175.394,45.900,159.356
C06791=1040.058,432.850,-142.220,175.408,45.908,159.359
C06792=1040.069,433.095,-142.270,175.422,45.916,159.363
C06793=1040.082,433.339,-142.321,175.435,45.924,159.367
C06794=1040.094,433.584,-142.372,175.450,45.932,159.371
C06795=1040.106,433.828,-142.423,175.464,45.940,159.375
C06796=1040.118,434.072,-142.474,175.477,45.948,159.379
C06797=1040.130,434.317,-142.524,175.492,45.956,159.383
C06798=1040.142,434.561,-142.575,175.507,45.964,159.387
C06799=1040.154,434.806,-142.626,175.520,45.972,159.390
C06800=1040.166,435.050,-142.677,175.535,45.980,159.394
C06801=1040.185,435.425,-142.755,175.557,45.993,159.401
C06802=1040.204,435.799,-142.834,175.579,46.005,159.407
C06803=1040.222,436.173,-142.913,175.602,46.018,159.413
C06804=1040.241,436.547,-142.991,175.624,46.031,159.419
C06805=1040.253,436.791,-143.042,175.639,46.039,159.423
C06806=1040.265,437.036,-143.095,175.654,46.047,159.427
C06807=1040.278,437.280,-143.146,175.669,46.056,159.431
C06808=1040.290,437.525,-143.197,175.683,46.064,159.435
C06809=1040.302,437.769,-143.249,175.698,46.072,159.440
C06810=1040.315,438.013,-143.302,175.713,46.081,159.444
C06811=1040.327,438.258,-143.353,175.728,46.089,159.448
C06812=1040.340,438.501,-143.405,175.743,46.098,159.452
C06813=1040.353,438.746,-143.457,175.758,46.107,159.456
C06814=1040.364,438.990,-143.508,175.774,46.115,159.461
C06815=1040.377,439.235,-143.561,175.789,46.124,159.465
C06816=1040.389,439.479,-143.613,175.804,46.133,159.469
C06817=1040.403,439.723,-143.665,175.820,46.141,159.473
C06818=1040.415,439.967,-143.717,175.835,46.150,159.478
C06819=1040.428,440.212,-143.770,175.850,46.158,159.482
C06820=1040.440,440.455,-143.822,175.866,46.167,159.486
C06821=1040.453,440.699,-143.875,175.881,46.176,159.491
C06822=1040.465,440.943,-143.927,175.897,46.185,159.495
C06823=1040.478,441.188,-143.979,175.913,46.194,159.500
C06824=1040.491,441.432,-144.033,175.929,46.202,159.504
C06825=1040.503,441.676,-144.085,175.944,46.211,159.508
C06826=1040.517,441.919,-144.137,175.960,46.220,159.513
C06827=1040.530,442.163,-144.191,175.977,46.229,159.517
C06828=1040.543,442.408,-144.243,175.992,46.238,159.522
C06829=1040.556,442.651,-144.296,176.009,46.247,159.526
C06830=1040.569,442.895,-144.349,176.025,46.256,159.531
C06831=1040.582,443.139,-144.402,176.041,46.265,159.536
C06832=1040.595,443.384,-144.455,176.057,46.274,159.540
C06833=1040.613,443.725,-144.530,176.080,46.287,159.546
C06834=1040.631,444.066,-144.604,176.103,46.300,159.553
C06835=1040.650,444.407,-144.678,176.126,46.312,159.560
C06836=1040.668,444.748,-144.753,176.150,46.325,159.566
C06837=1040.683,444.990,-144.806,176.166,46.334,159.571
C06838=1040.697,445.234,-144.858,176.183,46.343,159.575
C06839=1040.712,445.477,-144.910,176.200,46.352,159.580
C06840=1040.727,445.721,-144.961,176.217,46.361,159.585
C06841=1040.743,445.964,-145.012,176.234,46.369,159.589
C06842=1040.760,446.208,-145.062,176.251,46.378,159.594
C06843=1040.778,446.453,-145.112,176.268,46.387,159.598
C06844=1040.795,446.696,-145.162,176.286,46.395,159.603
C06845=1040.814,446.940,-145.211,176.303,46.403,159.607
C06846=1040.833,447.185,-145.260,176.320,46.411,159.612
C06847=1040.852,447.429,-145.307,176.337,46.419,159.616
C06848=1040.872,447.674,-145.356,176.356,46.427,159.621
C06849=1040.893,447.918,-145.403,176.373,46.435,159.625
C06850=1040.915,448.162,-145.450,176.391,46.443,159.630
C06851=1040.937,448.407,-145.496,176.408,46.451,159.634
C06852=1040.959,448.651,-145.541,176.426,46.458,159.639
C06853=1040.983,448.896,-145.587,176.444,46.465,159.643
C06854=1041.006,449.141,-145.632,176.462,46.472,159.647
C06855=1041.030,449.386,-145.676,176.480,46.480,159.652
C06856=1041.055,449.632,-145.720,176.499,46.487,159.656
C06857=1041.082,449.888,-145.765,176.518,46.494,159.660
C06858=1041.109,450.145,-145.811,176.538,46.501,159.665
C06859=1041.137,450.401,-145.854,176.557,46.509,159.670
C06860=1041.166,450.658,-145.898,176.576,46.516,159.674
C06861=1041.194,450.904,-145.940,176.595,46.523,159.678
C06862=1041.222,451.150,-145.981,176.613,46.529,159.683
C06863=1041.251,451.395,-146.022,176.632,46.535,159.687
C06864=1041.281,451.640,-146.062,176.651,46.542,159.691
C06865=1040.983,451.687,-146.379,176.654,46.619,159.715
C06866=1040.954,451.444,-146.339,176.635,46.612,159.710
C06867=1040.925,451.201,-146.299,176.616,46.606,159.706
C06868=1040.896,450.957,-146.258,176.598,46.600,159.702
C06869=1040.869,450.713,-146.217,176.579,46.594,159.698
C06870=1040.841,450.469,-146.176,176.561,46.586,159.693
C06871=1040.814,450.225,-146.134,176.542,46.580,159.689
C06872=1040.788,449.982,-146.091,176.523,46.573,159.685
C06873=1040.763,449.738,-146.049,176.505,46.566,159.681
C06874=1040.737,449.493,-146.006,176.488,46.559,159.676
C06875=1040.713,449.248,-145.961,176.469,46.552,159.672
C06876=1040.689,449.003,-145.916,176.450,46.545,159.667
C06877=1040.666,448.758,-145.871,176.432,46.538,159.663
C06878=1040.642,448.513,-145.826,176.414,46.530,159.659
C06879=1040.620,448.269,-145.780,176.397,46.523,159.654
C06880=1040.598,448.024,-145.733,176.379,46.515,159.650
C06881=1040.578,447.780,-145.686,176.361,46.508,159.646
C06882=1040.557,447.535,-145.638,176.344,46.500,159.641
C06883=1040.536,447.290,-145.590,176.325,46.492,159.636
C06884=1040.517,447.046,-145.543,176.308,46.484,159.632
C06885=1040.498,446.803,-145.494,176.291,46.475,159.627
C06886=1040.480,446.558,-145.445,176.273,46.467,159.623
C06887=1040.462,446.314,-145.395,176.256,46.459,159.618
C06888=1040.445,446.070,-145.345,176.239,46.451,159.614
C06889=1040.429,445.827,-145.294,176.222,46.442,159.609
C06890=1040.413,445.582,-145.243,176.205,46.434,159.605
C06891=1040.398,445.339,-145.191,176.188,46.425,159.600
C06892=1040.383,445.096,-145.139,176.170,46.416,159.595
C06893=1040.368,444.853,-145.086,176.154,46.407,159.591
C06894=1040.355,444.609,-145.033,176.138,46.398,159.586
C06895=1040.342,444.366,-144.981,176.121,46.389,159.582
C06896=1040.329,444.123,-144.927,176.104,46.380,159.577
C06897=1040.316,443.879,-144.874,176.088,46.371,159.572
C06898=1040.302,443.635,-144.821,176.071,46.362,159.568
C06899=1040.289,443.391,-144.767,176.054,46.353,159.563
C06900=1040.276,443.147,-144.714,176.038,46.344,159.558
C06901=1040.262,442.904,-144.662,176.023,46.335,159.554
C06902=1040.250,442.660,-144.609,176.006,46.326,159.549
C06903=1040.237,442.416,-144.556,175.990,46.317,159.545
C06904=1040.224,442.172,-144.503,175.973,46.308,159.540
C06905=1040.211,441.928,-144.450,175.958,46.300,159.536
C06906=1040.198,441.683,-144.397,175.942,46.290,159.531
C06907=1040.186,441.440,-144.345,175.925,46.282,159.527
C06908=1040.173,441.195,-144.292,175.910,46.273,159.522
C06909=1040.160,440.951,-144.239,175.894,46.264,159.518
C06910=1040.148,440.707,-144.187,175.879,46.256,159.514
C06911=1040.135,440.463,-144.134,175.863,46.247,159.509
C06912=1040.122,440.218,-144.082,175.847,46.238,159.505
C06913=1040.109,439.975,-144.029,175.831,46.230,159.501
C06914=1040.096,439.731,-143.977,175.816,46.221,159.496
C06915=1040.084,439.487,-143.925,175.800,46.213,159.492
C06916=1040.071,439.242,-143.872,175.785,46.204,159.488
C06917=1040.059,438.998,-143.821,175.770,46.195,159.483
C06918=1040.047,438.763,-143.770,175.755,46.187,159.479
C06919=1040.035,438.529,-143.721,175.741,46.179,159.475
C06920=1040.022,438.294,-143.671,175.726,46.171,159.471
C06921=1040.011,438.060,-143.622,175.711,46.163,159.467
C06922=1039.998,437.824,-143.571,175.697,46.155,159.463
C06923=1039.987,437.590,-143.522,175.683,46.147,159.459
C06924=1039.975,437.356,-143.472,175.668,46.139,159.455
C06925=1039.963,437.121,-143.422,175.654,46.131,159.451
C06926=1039.951,436.876,-143.371,175.639,46.122,159.447
C06927=1039.938,436.632,-143.319,175.624,46.114,159.443
C06928=1039.926,436.388,-143.268,175.609,46.106,159.439
C06929=1039.914,436.143,-143.216,175.595,46.098,159.435
C06930=1039.901,435.895,-143.164,175.580,46.089,159.431
C06931=1039.889,435.647,-143.112,175.565,46.081,159.427
C06932=1039.877,435.399,-143.060,175.551,46.073,159.423
C06933=1039.864,435.151,-143.008,175.536,46.065,159.419
C06934=1039.852,434.907,-142.956,175.521,46.057,159.415
C06935=1039.840,434.662,-142.906,175.507,46.049,159.411
C06936=1039.828,434.417,-142.855,175.492,46.041,159.407
C06937=1039.816,434.173,-142.804,175.479,46.032,159.403
C06938=1039.804,433.928,-142.753,175.464,46.025,159.399
C06939=1039.791,433.684,-142.703,175.450,46.017,159.395
C06940=1039.779,433.439,-142.652,175.436,46.009,159.391
C06941=1039.767,433.194,-142.601,175.422,46.001,159.387
C06942=1039.756,432.950,-142.551,175.408,45.993,159.384
C06943=1039.743,432.706,-142.500,175.394,45.985,159.380
C06944=1039.732,432.461,-142.449,175.380,45.977,159.376
C06945=1039.719,432.216,-142.399,175.366,45.970,159.372
C06946=1039.708,431.972,-142.348,175.353,45.962,159.369
C06947=1039.696,431.727,-142.298,175.338,45.955,159.365
C06948=1039.684,431.482,-142.247,175.325,45.946,159.361
C06949=1039.672,431.238,-142.198,175.312,45.939,159.357
C06950=1039.661,430.993,-142.147,175.298,45.931,159.354
C06951=1039.649,430.749,-142.097,175.285,45.923,159.350
C06952=1039.638,430.504,-142.047,175.270,45.916,159.346
C06953=1039.626,430.259,-141.997,175.257,45.908,159.342
C06954=1039.614,430.015,-141.947,175.244,45.901,159.339
C06955=1039.603,429.770,-141.896,175.231,45.893,159.335
C06956=1039.591,429.525,-141.847,175.217,45.886,159.332
C06957=1039.580,429.280,-141.797,175.204,45.878,159.328
C06958=1039.568,429.036,-141.747,175.191,45.870,159.324
C06959=1039.557,428.790,-141.697,175.178,45.863,159.321
C06960=1039.545,428.546,-141.647,175.165,45.855,159.317
C06961=1039.534,428.301,-141.598,175.151,45.848,159.314
C06962=1039.522,428.056,-141.548,175.138,45.841,159.310
C06963=1039.511,427.812,-141.499,175.125,45.833,159.307
C06964=1039.500,427.567,-141.449,175.112,45.826,159.303
C06965=1039.488,427.321,-141.400,175.099,45.819,159.300
C06966=1039.476,427.077,-141.350,175.087,45.811,159.296
C06967=1039.465,426.832,-141.301,175.074,45.804,159.293
C06968=1039.454,426.587,-141.251,175.061,45.796,159.289
C06969=1039.443,426.342,-141.202,175.048,45.790,159.286
C06970=1039.431,426.097,-141.153,175.035,45.782,159.282
C06971=1039.419,425.852,-141.104,175.023,45.775,159.279
C06972=1039.408,425.608,-141.055,175.010,45.768,159.276
C06973=1039.397,425.363,-141.005,174.998,45.761,159.272
C06974=1039.386,425.117,-140.957,174.985,45.753,159.269
C06975=1039.375,424.872,-140.908,174.973,45.746,159.266
C06976=1039.363,424.628,-140.859,174.960,45.740,159.262
C06977=1039.352,424.382,-140.811,174.948,45.732,159.259
C06978=1039.342,424.137,-140.761,174.936,45.725,159.256
C06979=1039.331,423.893,-140.712,174.923,45.718,159.252
C06980=1039.320,423.648,-140.664,174.911,45.711,159.249
C06981=1039.309,423.402,-140.616,174.898,45.704,159.246
C06982=1039.297,423.158,-140.567,174.887,45.697,159.242
C06983=1039.286,422.912,-140.518,174.874,45.691,159.239
C06984=1039.275,422.667,-140.470,174.862,45.684,159.236
C06985=1039.264,422.422,-140.421,174.850,45.677,159.233
C06986=1039.253,422.192,-140.376,174.839,45.670,159.230
C06987=1039.243,421.961,-140.330,174.828,45.664,159.227
C06988=1039.232,421.731,-140.285,174.816,45.658,159.224
C06989=1039.222,421.500,-140.241,174.805,45.652,159.221
C06990=1039.213,421.269,-140.195,174.794,45.645,159.218
C06991=1039.202,421.039,-140.150,174.782,45.638,159.215
C06992=1039.192,420.808,-140.104,174.772,45.632,159.212
C06993=1039.181,420.578,-140.059,174.761,45.626,159.209
C06994=1039.170,420.332,-140.011,174.749,45.619,159.206
C06995=1039.160,420.087,-139.963,174.737,45.612,159.203
C06996=1039.149,419.842,-139.915,174.726,45.606,159.200
C06997=1039.138,419.597,-139.867,174.714,45.599,159.197
C06998=1039.127,419.352,-139.819,174.702,45.593,159.194
C06999=1039.117,419.106,-139.772,174.691,45.586,159.191
C07000=1039.107,418.862,-139.724,174.680,45.579,159.187
C07001=1039.096,418.616,-139.676,174.667,45.573,159.184
C07002=1039.085,418.371,-139.628,174.656,45.566,159.181
C07003=1039.074,418.125,-139.581,174.645,45.559,159.178
C07004=1039.064,417.880,-139.533,174.634,45.553,159.175
C07005=1039.053,417.635,-139.486,174.622,45.547,159.172
C07006=1039.042,417.389,-139.439,174.611,45.540,159.169
C07007=1039.032,417.144,-139.391,174.600,45.534,159.167
C07008=1039.021,416.900,-139.344,174.589,45.527,159.163
C07009=1039.010,416.654,-139.296,174.578,45.521,159.161
C07010=1039.000,416.409,-139.249,174.567,45.515,159.158
C07011=1038.989,416.164,-139.203,174.556,45.508,159.155
C07012=1038.979,415.918,-139.155,174.544,45.502,159.152
C07013=1038.969,415.673,-139.108,174.533,45.496,159.149
C07014=1038.958,415.427,-139.061,174.522,45.490,159.146
C07015=1038.947,415.182,-139.014,174.511,45.484,159.143
C07016=1038.937,414.936,-138.967,174.500,45.477,159.140
C07017=1038.927,414.691,-138.920,174.489,45.471,159.137
C07018=1038.916,414.446,-138.874,174.478,45.465,159.135
C07019=1038.906,414.201,-138.826,174.467,45.458,159.132
C07020=1038.896,413.955,-138.780,174.456,45.453,159.129
C07021=1038.885,413.710,-138.733,174.446,45.447,159.126
C07022=1038.875,413.464,-138.686,174.436,45.440,159.124
C07023=1038.865,413.219,-138.639,174.425,45.434,159.121
C07024=1038.854,412.974,-138.593,174.414,45.428,159.118
C07025=1038.844,412.728,-138.546,174.403,45.422,159.115
C07026=1038.833,412.483,-138.500,174.392,45.416,159.112
C07027=1038.824,412.238,-138.454,174.382,45.410,159.110
C07028=1038.814,411.992,-138.407,174.372,45.404,159.107
C07029=1038.803,411.747,-138.361,174.361,45.398,159.104
C07030=1038.793,411.501,-138.314,174.350,45.392,159.101
C07031=1038.782,411.255,-138.268,174.340,45.386,159.099
C07032=1038.772,411.009,-138.222,174.329,45.380,159.096
C07033=1038.762,410.764,-138.176,174.319,45.374,159.093
C07034=1038.752,410.519,-138.130,174.309,45.368,159.091
C07035=1038.742,410.273,-138.084,174.298,45.363,159.088
C07036=1038.731,410.027,-138.038,174.289,45.357,159.086
C07037=1038.721,409.782,-137.992,174.278,45.351,159.083
C07038=1038.711,409.536,-137.946,174.267,45.345,159.080
C07039=1038.701,409.291,-137.900,174.258,45.339,159.078
C07040=1038.690,409.045,-137.855,174.247,45.334,159.075
C07041=1038.681,408.799,-137.808,174.237,45.328,159.072
C07042=1038.671,408.554,-137.763,174.227,45.322,159.070
C07043=1038.661,408.309,-137.717,174.217,45.317,159.067
C07044=1038.651,408.062,-137.671,174.207,45.311,159.065
C07045=1038.640,407.817,-137.625,174.197,45.305,159.062
C07046=1038.631,407.590,-137.583,174.187,45.300,159.060
C07047=1038.622,407.364,-137.542,174.178,45.295,159.058
C07048=1038.613,407.137,-137.500,174.169,45.289,159.055
C07049=1038.604,406.911,-137.457,174.160,45.285,159.053
C07050=1038.595,406.685,-137.415,174.151,45.279,159.051
C07051=1038.586,406.458,-137.374,174.142,45.274,159.048
C07052=1038.577,406.232,-137.332,174.132,45.269,159.046
C07053=1038.568,406.005,-137.289,174.123,45.264,159.044
C07054=1038.558,405.760,-137.245,174.114,45.258,159.041
C07055=1038.548,405.514,-137.200,174.105,45.253,159.039
C07056=1038.539,405.268,-137.154,174.094,45.248,159.036
C07057=1038.529,405.023,-137.108,174.085,45.241,159.034
C07058=1038.519,404.777,-137.064,174.076,45.236,159.031
C07059=1038.509,404.532,-137.019,174.065,45.231,159.029
C07060=1038.500,404.285,-136.973,174.056,45.225,159.026
C07061=1038.490,404.040,-136.928,174.047,45.220,159.024
C07062=1038.480,403.794,-136.883,174.036,45.215,159.022
C07063=1038.471,403.549,-136.838,174.027,45.209,159.019
C07064=1038.461,403.303,-136.793,174.018,45.204,159.017
C07065=1038.452,403.058,-136.748,174.009,45.198,159.014
C07066=1038.441,402.811,-136.703,173.998,45.193,159.012
C07067=1038.432,402.566,-136.658,173.989,45.188,159.010
C07068=1038.422,402.320,-136.614,173.980,45.182,159.007
C07069=1038.413,402.074,-136.569,173.971,45.177,159.005
C07070=1038.403,401.829,-136.525,173.961,45.172,159.003
C07071=1038.393,401.582,-136.480,173.951,45.167,159.000
C07072=1038.384,401.337,-136.435,173.942,45.162,158.998
C07073=1038.375,401.091,-136.390,173.933,45.156,158.996
C07074=1038.365,400.845,-136.346,173.924,45.151,158.993
C07075=1038.356,400.600,-136.301,173.915,45.146,158.991
C07076=1038.346,400.353,-136.257,173.906,45.141,158.989
C07077=1038.336,400.108,-136.213,173.896,45.136,158.986
C07078=1038.326,399.862,-136.169,173.887,45.131,158.984
C07079=1038.318,399.617,-136.125,173.877,45.125,158.982
C07080=1038.308,399.371,-136.080,173.869,45.121,158.980
C07081=1038.298,399.125,-136.036,173.860,45.116,158.977
C07082=1038.289,398.879,-135.992,173.851,45.111,158.975
C07083=1038.280,398.633,-135.948,173.842,45.106,158.973
C07084=1038.270,398.387,-135.904,173.833,45.101,158.971
C07085=1038.260,398.142,-135.860,173.823,45.095,158.968
C07086=1038.251,397.896,-135.816,173.814,45.090,158.966
C07087=1038.242,397.650,-135.772,173.805,45.085,158.964
C07088=1038.232,397.404,-135.728,173.797,45.080,158.962
C07089=1038.223,397.158,-135.684,173.788,45.076,158.960
C07090=1038.214,396.912,-135.640,173.779,45.071,158.957
C07091=1038.204,396.666,-135.596,173.770,45.066,158.955
C07092=1038.195,396.420,-135.553,173.761,45.061,158.953
C07093=1038.186,396.174,-135.509,173.752,45.056,158.951
C07094=1038.176,395.928,-135.465,173.744,45.051,158.949
C07095=1038.168,395.683,-135.421,173.735,45.046,158.947
C07096=1038.158,395.437,-135.378,173.726,45.042,158.945
C07097=1038.149,395.191,-135.335,173.717,45.037,158.943
C07098=1038.140,394.944,-135.291,173.709,45.032,158.940
C07099=1038.131,394.699,-135.247,173.700,45.028,158.938
C07100=1038.121,394.453,-135.204,173.691,45.023,158.936
C07101=1038.112,394.207,-135.160,173.683,45.018,158.934
C07102=1038.103,393.960,-135.117,173.674,45.013,158.932
C07103=1038.093,393.715,-135.073,173.666,45.009,158.930
C07104=1038.084,393.469,-135.030,173.657,45.004,158.928
C07105=1038.075,393.223,-134.987,173.648,44.999,158.926
C07106=1038.068,393.006,-134.949,173.641,44.995,158.924
C07107=1038.059,392.790,-134.911,173.633,44.991,158.922
C07108=1038.051,392.573,-134.873,173.626,44.987,158.920
C07109=1038.043,392.357,-134.835,173.618,44.983,158.919
C07110=1038.035,392.140,-134.796,173.611,44.979,158.917
C07111=1038.028,391.924,-134.759,173.604,44.975,158.915
C07112=1038.019,391.707,-134.721,173.596,44.971,158.913
C07113=1038.011,391.491,-134.683,173.589,44.967,158.912
C07114=1038.002,391.245,-134.641,173.580,44.962,158.910
C07115=1037.993,390.998,-134.597,173.573,44.958,158.908
C07116=1037.984,390.752,-134.555,173.564,44.953,158.906
C07117=1037.975,390.506,-134.512,173.555,44.949,158.904
C07118=1037.966,390.261,-134.469,173.548,44.944,158.902
C07119=1037.957,390.014,-134.426,173.539,44.940,158.900
C07120=1037.947,389.768,-134.383,173.531,44.935,158.898
C07121=1037.939,389.522,-134.340,173.523,44.931,158.896
C07122=1037.930,389.276,-134.298,173.514,44.926,158.894
C07123=1037.921,389.030,-134.255,173.507,44.922,158.892
C07124=1037.912,388.783,-134.213,173.498,44.918,158.890
C07125=1037.903,388.537,-134.170,173.490,44.913,158.888
C07126=1037.894,388.291,-134.127,173.482,44.908,158.886
C07127=1037.885,388.046,-134.085,173.473,44.905,158.884
C07128=1037.877,387.799,-134.043,173.466,44.900,158.882
C07129=1037.867,387.553,-134.000,173.457,44.896,158.880
C07130=1037.858,387.307,-133.959,173.450,44.891,158.878
C07131=1037.849,387.060,-133.915,173.441,44.888,158.877
C07132=1037.840,386.814,-133.873,173.434,44.883,158.875
C07133=1037.831,386.568,-133.831,173.425,44.879,158.873
C07134=1037.822,386.322,-133.789,173.417,44.874,158.871
C07135=1037.813,386.076,-133.747,173.409,44.870,158.869
C07136=1037.804,385.830,-133.705,173.402,44.866,158.867
C07137=1037.796,385.583,-133.663,173.393,44.862,158.865
C07138=1037.787,385.337,-133.620,173.386,44.858,158.864
C07139=1037.778,385.091,-133.579,173.378,44.854,158.862
C07140=1037.769,384.844,-133.537,173.370,44.850,158.860
C07141=1037.760,384.598,-133.495,173.362,44.845,158.858
C07142=1037.751,384.352,-133.452,173.354,44.841,158.856
C07143=1037.742,384.106,-133.411,173.347,44.837,158.854
C07144=1037.734,383.860,-133.369,173.339,44.833,158.853
C07145=1037.725,383.614,-133.327,173.331,44.829,158.851
C07146=1037.716,383.367,-133.286,173.324,44.825,158.849
C07147=1037.707,383.121,-133.244,173.315,44.821,158.847
C07148=1037.699,382.874,-133.202,173.308,44.817,158.845
C07149=1037.690,382.628,-133.160,173.300,44.813,158.844
C07150=1037.682,382.382,-133.119,173.292,44.809,158.842
C07151=1037.673,382.136,-133.077,173.285,44.805,158.840
C07152=1037.664,381.889,-133.035,173.277,44.800,158.838
C07153=1037.655,381.643,-132.993,173.270,44.796,158.837
C07154=1037.647,381.397,-132.953,173.262,44.792,158.835
C07155=1037.639,381.150,-132.911,173.255,44.789,158.833
C07156=1037.630,380.904,-132.869,173.247,44.785,158.831
C07157=1037.621,380.658,-132.827,173.240,44.781,158.830
C07158=1037.613,380.411,-132.786,173.231,44.777,158.828
C07159=1037.604,380.165,-132.745,173.224,44.773,158.826
C07160=1037.596,379.919,-132.703,173.217,44.769,158.825
C07161=1037.588,379.672,-132.662,173.210,44.765,158.823
C07162=1037.579,379.425,-132.620,173.203,44.761,158.821
C07163=1037.570,379.180,-132.579,173.194,44.757,158.819
C07164=1037.562,378.933,-132.538,173.187,44.753,158.818
C07165=1037.553,378.687,-132.496,173.180,44.750,158.816
C07166=1037.539,378.288,-132.430,173.168,44.743,158.813
C07167=1037.525,377.890,-132.364,173.156,44.737,158.811
C07168=1037.512,377.492,-132.297,173.144,44.731,158.808
C07169=1037.497,377.092,-132.231,173.133,44.725,158.805
C07170=1037.489,376.846,-132.191,173.125,44.722,158.804
C07171=1037.481,376.599,-132.149,173.117,44.718,158.802
C07172=1037.472,376.353,-132.108,173.110,44.714,158.800
C07173=1037.464,376.106,-132.067,173.103,44.710,158.799
C07174=1037.455,375.860,-132.027,173.096,44.707,158.797
C07175=1037.446,375.613,-131.986,173.089,44.703,158.796
C07176=1037.438,375.367,-131.946,173.082,44.700,158.794
C07177=1037.430,375.121,-131.905,173.075,44.696,158.792
C07178=1037.422,374.874,-131.864,173.068,44.692,158.791
C07179=1037.413,374.628,-131.824,173.060,44.688,158.789
C07180=1037.404,374.381,-131.783,173.053,44.685,158.788
C07181=1037.396,374.134,-131.742,173.046,44.681,158.786
C07182=1037.388,373.888,-131.702,173.039,44.678,158.784
C07183=1037.379,373.641,-131.661,173.032,44.674,158.783
C07184=1037.371,373.395,-131.621,173.025,44.670,158.781
C07185=1037.363,373.148,-131.581,173.018,44.667,158.780
C07186=1037.355,372.902,-131.540,173.011,44.664,158.778
C07187=1037.347,372.655,-131.499,173.004,44.660,158.777
C07188=1037.338,372.409,-131.459,172.997,44.656,158.775
C07189=1037.330,372.162,-131.419,172.990,44.653,158.774
C07190=1037.322,371.916,-131.378,172.983,44.649,158.772
C07191=1037.313,371.669,-131.337,172.976,44.646,158.771
C07192=1037.305,371.422,-131.298,172.969,44.643,158.769
C07193=1037.297,371.176,-131.258,172.962,44.639,158.767
C07194=1037.289,370.929,-131.218,172.955,44.636,158.766
C07195=1037.281,370.683,-131.177,172.948,44.632,158.764
